METHOD PRIVATE Meth_MororON : BOOL
VAR_INPUT
	Execute: 	BOOL;
END_VAR


	THIS^.Monitoring.StepMessage			:= 'Motor ON';
	THIS^.Monitoring.Error_Text				:= ' Motor ON Fail';
	//THIS^.CMD.Deacivate_Sequence_Time_Out	:= TRUE;	// Disable time out to the all sequence
	THIS^.CMD.DeactivateStepTimeOut			:= TRUE;	// Disable time out to the actual step
	THIS^.Parameter.TimeOut					:= T#5S;


											
	THIS^.Delay.IN:=TRUE;
	THIS^.Delay.PT :=DINT_TO_TIME( Persist.PersistentStruct.TimerMotorOn);// Ctrl_ref.Parameters.TimerPressDown1);
	IF THIS^.Delay.Q  AND FB_RW_Ctrl_ref.Done THEN
		Meth_MororON	:= TRUE;
	END_IF
END_METHOD

METHOD Meth_OutGripperClamp : BOOL
VAR_INPUT
	Execute: 	BOOL;
END_VAR


	THIS^.Monitoring.StepMessage			:= 'Output Gripper Close';
	THIS^.Monitoring.Error_Text				:= ' Fail';
	//THIS^.CMD.Deacivate_Sequence_Time_Out	:= TRUE;	// Disable time out to the all sequence
	THIS^.CMD.DeactivateStepTimeOut			:= TRUE;	// Disable time out to the actual step
	THIS^.Parameter.TimeOut					:= T#5S;

	gMachineCtrl.IO.Out.Output_GripperClose:=TRUE;
											
	THIS^.Delay.IN:=TRUE;
	THIS^.Delay.PT :=DINT_TO_TIME( Persist.PersistentStruct.TimeOutputGripperClose);// Ctrl_ref.Parameters.TimerPressDown1);
	IF THIS^.Delay.Q THEN
		Meth_OutGripperClamp	:= TRUE;
		
		//gMachineCtrl.Parameters.UW_1_Param.EnableTension:=TRUE;
		//gMachineCtrl.Parameters.UW_2_Param.EnableTension:=TRUE;
		
	END_IF
END_METHOD

METHOD Meth_OutGripperEndPos : BOOL
VAR_INPUT
	Execute: 	BOOL;
END_VAR
VAR_INST
	ExecuteTrig: 	Trigger;
END_VAR




IF ExecuteTrig.EDGEPOS(Execute) THEN
	Meth_OutGripperEndPos:=	FALSE;
	THIS^.SubStepNo:= 	1;	
END_IF

IF ExecuteTrig.EDGENEG(Execute) THEN
	Meth_OutGripperEndPos:=	FALSE;
END_IF

CASE THIS^.SubStepNo OF
	(* Power ON*)
	1:
		THIS^.Monitoring.StepMessage	:= 'Move output gripper to end';								
		gWebAxes.Output.Crtl.Basic_axis.Input.Command.MoveAbsolute		:= TRUE;
		gWebAxes.Output.Crtl.Basic_axis.Input.Parameter.Velocity		:= 500;//mm/sec
		gWebAxes.Output.Crtl.Basic_axis.Input.Parameter.Position		:= gMachineCtrl.Parameters.OutgripperEndPosition;//mm
		
		THIS^.SubStepNo:= 2;		
	
	2:	
		THIS^.Monitoring.StepMessage:= 'Wait output gripper end';
		
		IF gWebAxes.Output.Crtl.Basic_axis.Output.monitor.ActPosition > (gMachineCtrl.Parameters.OutgripperEndPosition-200) THEN
			gMachineCtrl.IO.Out.Output_GripperClose:=FALSE;
		END_IF
							
		IF gWebAxes.Output.Crtl.Basic_axis.Output.Status.MC_MoveAbsolut.Done THEN
			THIS^.SubStepNo	:= 3 ;
		END_IF
		
	3:	
		THIS^.Monitoring.StepMessage	:= 'Move output gripper to end';								
		gWebAxes.Output.Crtl.Basic_axis.Input.Command.MoveAbsolute		:= TRUE;
		gWebAxes.Output.Crtl.Basic_axis.Input.Parameter.Velocity		:= 100;//mm/sec
		gWebAxes.Output.Crtl.Basic_axis.Input.Parameter.Position		:= gMachineCtrl.Parameters.OutgripperEndPosition+200;//mm
		
		THIS^.SubStepNo:= 4;	
				
	4:	
		THIS^.Monitoring.StepMessage:= 'Wait output gripper end';
							
		IF gWebAxes.Output.Crtl.Basic_axis.Output.Status.MC_MoveAbsolut.Done THEN
			THIS^.SubStepNo	:= 100 ;
			Meth_OutGripperEndPos:=	TRUE;
		END_IF							
END_CASE
END_METHOD

METHOD Meth_OutGripperStartPos : BOOL
VAR_INPUT
	Execute: 	BOOL;
END_VAR
VAR_INST
	ExecuteTrig: 	Trigger;
END_VAR




IF ExecuteTrig.EDGEPOS(Execute) THEN
	Meth_OutGripperStartPos:=	FALSE;
	THIS^.SubStepNo:= 	1;	
END_IF

IF ExecuteTrig.EDGENEG(Execute) THEN
	Meth_OutGripperStartPos:=	FALSE;
END_IF

CASE THIS^.SubStepNo OF
	(* Power ON*)
	1:
		THIS^.Monitoring.StepMessage	:= 'Move output gripper to home';								
		gWebAxes.Output.Crtl.Basic_axis.Input.Command.MoveAbsolute		:= TRUE;
		gWebAxes.Output.Crtl.Basic_axis.Input.Parameter.Velocity		:= 500;//mm/sec
		gWebAxes.Output.Crtl.Basic_axis.Input.Parameter.Position		:= 0;
		
		THIS^.SubStepNo:= 2;		
	
	2:	
		THIS^.Monitoring.StepMessage:= 'Wait output gripper home';
									
		IF gWebAxes.Output.Crtl.Basic_axis.Output.Status.MC_MoveAbsolut.Done THEN
			THIS^.SubStepNo	:= 3 ;
			Meth_OutGripperStartPos	:= TRUE;
		END_IF
		

							
END_CASE
END_METHOD

METHOD Meth_Rest_IO 
VAR_INPUT
	
END_VAR

Ctrl_ref.IO.Out.HeaterOn := FALSE;
END_METHOD

METHOD PRIVATE Meth_WaitDancerFull : BOOL
VAR_INPUT
	Execute: 	BOOL;
END_VAR


	//THIS^.Monitoring.StepMessage			:= 'Gripper Retract';
	THIS^.Monitoring.Error_Text				:= ' Fail';
	//THIS^.CMD.Deacivate_Sequence_Time_Out	:= TRUE;	// Disable time out to the all sequence
	THIS^.CMD.DeactivateStepTimeOut			:= TRUE;	// Disable time out to the actual step
	THIS^.Parameter.TimeOut					:= T#5S;

	gMachineCtrl.Parameters.UW_1_Param.EnableDancer :=TRUE;
	gMachineCtrl.Parameters.UW_2_Param.EnableDancer:=TRUE;
											
	THIS^.Delay.IN:=TRUE;
	THIS^.Delay.PT :=DINT_TO_TIME( Persist.PersistentStruct.TimeGripperRetract);// Ctrl_ref.Parameters.TimerPressDown1);
	IF  (gMachineCtrl.Status.UW_1_DancerFull 
	AND gMachineCtrl.Status.UW_2_DancerFull)
	OR gMachineCtrl.Simulation THEN
		Meth_WaitDancerFull	:= TRUE;
	END_IF
END_METHOD

END_FUNCTION_BLOCK

// ---- POUs/App/FB_HeaterProtection.TcPOU
FUNCTION_BLOCK FB_HeaterProtection
VAR_INPUT
	Excute:BOOL;
END_VAR
VAR_OUTPUT
	Done:BOOL;
	Busy:BOOL;
END_VAR
VAR
	Timer:TON;
	Step:INT;
END_VAR


IF Excute THEN
	Step:= 10;
	Done:=FALSE;
	Excute:=FALSE;
	Busy:=TRUE;
	
	
END_IF

CASE Step OF

	0://wait
	
	10:
		Timer.PT := DINT_TO_TIME( Persist.PersistentStruct.TimerHotWeldingOn);
		Timer.IN:=TRUE;
		gMachineCtrl.IO.Out.HeaterOn:=TRUE;
		IF Timer.Q THEN
			gMachineCtrl.IO.Out.HeaterOn:=FALSE;
			Step:=20;
		END_IF
	
	20:
		Done:=TRUE;
		Timer.IN:=FALSE;
		Busy:=FALSE;
	
END_CASE

Timer();

END_FUNCTION_BLOCK

// ---- POUs/App/FB_Mechinit.TcPOU
FUNCTION_BLOCK FB_Mechinit EXTENDS CycleHandleFB
VAR_INPUT
	Ctrl_ref:			REFERENCE TO Ctrl_Typ;
END_VAR
VAR_OUTPUT
END_VAR
VAR
	MethInitDone:		BOOL;
END_VAR

VAR CONSTANT
// States are global
		
	MECHINIT_INIT:							INT:=0;
	MECHINIT_SWITCH_ON:						INT:=10;
	MECHINIT_RUN_MASTER:					INT:=20;
	MECHINIT_GEAR_IN:						INT:=30;
	MECHINIT_DONE:							INT:=100;
END_VAR

	IF NOT MethInitDone THEN
		MethInitDone	:= Meth_Init();
	END_IF
	
	IF  THIS^.CMD.Pause = FALSE THEN
		
		//-----------------------------
		//State Machine
		//-----------------------------
		CASE THIS^.StepNo OF
			MECHINIT_INIT:
				IF THIS^.StepOneShotTrig THEN
					THIS^.Monitoring.StepMessage	:= 'Init: Start.';
					THIS^.Delay(IN:=FALSE);
				ELSIF Meth_Enable(TRUE) THEN
					THIS^.StepNo	:= 	MECHINIT_SWITCH_ON;
				END_IF
			
			MECHINIT_SWITCH_ON:
				IF THIS^.StepOneShotTrig THEN
					THIS^.Monitoring.StepMessage	:= 'Switch motor on.';
					THIS^.Delay(IN:=FALSE);
					Meth_SwitchOn(FALSE);
				ELSIF Meth_SwitchOn(TRUE) THEN
					THIS^.StepNo	:= 	MECHINIT_RUN_MASTER;
				END_IF	
				
			MECHINIT_RUN_MASTER:
				IF THIS^.StepOneShotTrig THEN
					THIS^.Monitoring.StepMessage	:= 'Start master';
					THIS^.Delay(IN:=FALSE);
					Meth_StartVmaster(FALSE);
				ELSIF Meth_StartVmaster(TRUE) THEN
					THIS^.StepNo	:= 	MECHINIT_GEAR_IN;
				END_IF				
				

			MECHINIT_GEAR_IN:
				IF THIS^.StepOneShotTrig THEN
					THIS^.Monitoring.StepMessage	:= 'Gear In';
					THIS^.Delay(IN:=FALSE);
					Meth_GearIn(FALSE);
				ELSIF Meth_GearIn(TRUE) THEN
					THIS^.StepNo	:= 	MECHINIT_DONE;
				END_IF	
				
				
			MECHINIT_DONE:
				IF THIS^.StepOneShotTrig THEN
					THIS^.Monitoring.StepMessage	:= 'mechinit cycle Done';
				ELSIF Meth_Done(TRUE) THEN
					THIS^.StepNo	:= 	MECHINIT_INIT;
				END_IF					
				
		END_CASE
	
	ELSE
		THIS^.Monitoring.StepMessage:= 'Pause';
		
		IF THIS^.Status.Fault = TRUE THEN
		//IF Meth_EmStop(TRUE) THEN
				THIS^.CMD.ResetCycle	:= TRUE;		// Reset the all state machine to start point
		//END_IF
			
		END_IF
		
	END_IF
	
	THIS^.Delay();
	THIS^.CH_Logic();
	
	// Reset Meth_EmStop when at Init State
	IF THIS^.Pause = FALSE THEN
		//Meth_EmStop(FALSE);
	END_IF

METHOD PRIVATE Meth_Done : BOOL
VAR_INPUT
	Execute: 	BOOL;
END_VAR


	//THIS^.Monitoring.StepMessage			:= 'Press 1 engage';
	//THIS^.Monitoring.Error_Text				:= 'Press 1 engage Fail';
	//THIS^.CMD.Deacivate_Sequence_Time_Out	:= TRUE;	// Disable time out to the all sequence
	//THIS^.CMD.DeactivateStepTimeOut			:= TRUE;	// Disable time out to the actual step
	//THIS^.Parameter.TimeOut					:= T#5S;

	THIS^.Status.Done		:= TRUE;
	THIS^.Status.Running	:= FALSE;									
	Meth_Done	:= TRUE;
END_METHOD

METHOD PRIVATE Meth_Enable : BOOL
VAR_INPUT
	Execute: 	BOOL;
END_VAR


IF THIS^.CMD.Start THEN
	
	THIS^.Monitoring.StepMessage			:= 'Start';
	THIS^.Monitoring.Error_Text				:= 'Start Fail';
	THIS^.CMD.Deacivate_Sequence_Time_Out	:= TRUE;	// Disable time out to the all sequence
	THIS^.CMD.DeactivateStepTimeOut			:= TRUE;	// Disable time out to the actual step
	THIS^.Parameter.TimeOut					:= T#0.5S;

	THIS^.CMD.Start			:= FALSE;
	THIS^.Status.Done		:= FALSE;
	THIS^.Status.Running	:= TRUE;
	
	// Reset Commands and Statuses												
	
	Meth_Enable	:= TRUE;
END_IF
END_METHOD

METHOD Meth_GearIn : BOOL
VAR_INPUT
	Execute: 	BOOL;
END_VAR
VAR_INST	
	ExecuteTrig: 	Trigger;	
END_VAR
IF ExecuteTrig.EDGEPOS(Execute) THEN
	Meth_GearIn	:= FALSE;
	THIS^.SubStepNo:= 	1;	
END_IF

IF ExecuteTrig.EDGENEG(Execute) THEN
	Meth_GearIn	:=	FALSE;
END_IF

CASE THIS^.SubStepNo OF
	   
	1:
		THIS^.Monitoring.StepMessage:= 'Set GearInMultiMaster command';
		
		gWebAxes.UW_1.Crtl.MultiAxis.Input.Parameter.GearInMultiMaster.GearRatio1:=	0;

		
		gWebAxes.UW_1.Crtl.MultiAxis.Input.Parameter.GearInMultiMaster.Acceleration:= 	600000;
		gWebAxes.UW_1.Crtl.MultiAxis.Input.Parameter.GearInMultiMaster.Deceleration:= 	600000;
		gWebAxes.UW_1.Crtl.MultiAxis.Input.Parameter.GearInMultiMaster.Jerk:=			0;
		gWebAxes.UW_1.Crtl.MultiAxis.Input.Parameter.GearInMultiMaster.Options.AdvancedSlaveDynamics:= 	FALSE;
		
		gWebAxes.UW_1.Crtl.MultiAxis.Input.Command.GearInMultiMaster.StartSlave:=		TRUE;
				
								
		THIS^.SubStepNo	:= 2;		
			
	2:	
		THIS^.Monitoring.StepMessage:= 	'Wait for GearInMultiMaster done UW1' ;
							
		IF (gWebAxes.UW_1.Crtl.MultiAxis.Input.Command.GearInMultiMaster.StartSlave = FALSE) 
			AND (gWebAxes.UW_1.Crtl.MultiAxis.Output.Status.GearInMultiMaster.InGear = TRUE) THEN
			THIS^.SubStepNo:=	3;
		ELSIF 	gWebAxes.UW_1.Crtl.MultiAxis.Output.Status.GearInMultiMaster.InGear = TRUE THEN
			THIS^.SubStepNo:=	3;
		END_IF		


	3:
		THIS^.Monitoring.StepMessage:= 'Set GearInMultiMaster UW2 command';
		
		gWebAxes.UW_2.Crtl.MultiAxis.Input.Parameter.GearInMultiMaster.GearRatio1:=	0;

		
		gWebAxes.UW_2.Crtl.MultiAxis.Input.Parameter.GearInMultiMaster.Acceleration:= 	600000;
		gWebAxes.UW_2.Crtl.MultiAxis.Input.Parameter.GearInMultiMaster.Deceleration:= 	600000;
		gWebAxes.UW_2.Crtl.MultiAxis.Input.Parameter.GearInMultiMaster.Jerk:=			0;
		gWebAxes.UW_2.Crtl.MultiAxis.Input.Parameter.GearInMultiMaster.Options.AdvancedSlaveDynamics:= 	FALSE;
		
		gWebAxes.UW_2.Crtl.MultiAxis.Input.Command.GearInMultiMaster.StartSlave:=		TRUE;
				
								
		THIS^.SubStepNo	:= 4;		
			
	4:	
		THIS^.Monitoring.StepMessage:= 	'Wait for GearInMultiMaster done' ;
							
		IF (gWebAxes.UW_2.Crtl.MultiAxis.Input.Command.GearInMultiMaster.StartSlave = FALSE) 
			AND (gWebAxes.UW_2.Crtl.MultiAxis.Output.Status.GearInMultiMaster.InGear = TRUE) THEN
			THIS^.SubStepNo:=	0;
			Meth_GearIn:= 	TRUE;
		ELSIF gWebAxes.UW_2.Crtl.MultiAxis.Output.Status.GearInMultiMaster.InGear = TRUE THEN	
			THIS^.SubStepNo:=	0;
			Meth_GearIn:= 	TRUE;
		END_IF	

							
END_CASE
END_METHOD

METHOD Meth_Init :BOOL
VAR_INPUT
END_VAR
//resets


Meth_Init:=TRUE;
END_METHOD

METHOD Meth_StartVmaster : BOOL
VAR_INPUT
	Execute: 	BOOL;
END_VAR
VAR_INST	
	ExecuteTrig: 	Trigger;	
END_VAR

IF ExecuteTrig.EDGEPOS(Execute) THEN
	Meth_StartVmaster	:= FALSE;
	THIS^.SubStepNo:= 	1;	
END_IF

IF ExecuteTrig.EDGENEG(Execute) THEN
	Meth_StartVmaster	:=	FALSE;
END_IF


CASE THIS^.SubStepNo OF
	   
	1:
		THIS^.Monitoring.StepMessage	:= 'Set RunVel command to Master Tension';
		
			gWebAxes.UwVmaster.Crtl.Basic_axis.Input.Parameter.Acceleration	:= 100000; 
			gWebAxes.UwVmaster.Crtl.Basic_axis.Input.Parameter.Deceleration	:= 100000; 
			gWebAxes.UwVmaster.Crtl.Basic_axis.Input.Parameter.Velocity		:= 360000;//100000 
			gWebAxes.UwVmaster.Crtl.Basic_axis.Input.Parameter.Direction		:= MC_Positive_Direction; 		
				
			gWebAxes.UwVmaster.Crtl.Basic_axis.Input.Command.MoveVelocity		:= TRUE;
			THIS^.SubStepNo:= 	2;	

	2:	
		THIS^.Monitoring.StepMessage	:= 'Wait @ velocity from Master';
		IF (gWebAxes.UwVmaster.Crtl.Basic_axis.Output.Status.AxisStatus.ContinuousMotion = TRUE) THEN	
			Meth_StartVmaster:=TRUE;
			THIS^.SubStepNo:= 	0;				
		END_IF
								
END_CASE
END_METHOD

METHOD Meth_SwitchOn : BOOL
VAR_INPUT
	Execute: 	BOOL;
END_VAR
VAR_INST
	ExecuteTrig: 	Trigger;
END_VAR


IF ExecuteTrig.EDGEPOS(Execute) THEN
	Meth_SwitchOn:=	FALSE;
	THIS^.SubStepNo:= 	1;	
END_IF

IF ExecuteTrig.EDGENEG(Execute) THEN
	Meth_SwitchOn:=	FALSE;
END_IF

CASE THIS^.SubStepNo OF
	(* Power ON*)
	1:
		THIS^.Monitoring.StepMessage	:= 'Power On';								
		gWebAxes.UW_1.Crtl.Basic_axis.Input.Command.Power		:= TRUE;
		gWebAxes.UW_2.Crtl.Basic_axis.Input.Command.Power		:= TRUE;	
		gWebAxes.UwVmaster.Crtl.Basic_axis.Input.Command.Power	:= TRUE;
		
		THIS^.SubStepNo:= 2;		
	
	2:	
		THIS^.Monitoring.StepMessage:= 'Wait for standstill UW 1';
									
		IF gWebAxes.UW_1.Crtl.Basic_axis.Output.Status.AxisStatus.StandStill
		OR gWebAxes.UW_1.Crtl.Basic_axis.Output.Status.AxisStatus.SynchronizedMotion THEN
			THIS^.SubStepNo	:= 3 ;
		END_IF
		
	3:	
		THIS^.Monitoring.StepMessage:= 'Wait for standstill UW 2';
									
		IF gWebAxes.UW_2.Crtl.Basic_axis.Output.Status.AxisStatus.StandStill
		OR  gWebAxes.UW_2.Crtl.Basic_axis.Output.Status.AxisStatus.SynchronizedMotion THEN
			THIS^.SubStepNo	:= 4 ;
		END_IF		
		
	4:	
		THIS^.Monitoring.StepMessage:= 'Wait for standstill from master';
									
		IF gWebAxes.UwVmaster.Crtl.Basic_axis.Output.Status.AxisStatus.StandStill
		OR  gWebAxes.UwVmaster.Crtl.Basic_axis.Output.Status.AxisStatus.ContinuousMotion THEN
			THIS^.SubStepNo	:= 10 ;
			Meth_SwitchOn	:= TRUE;
		END_IF
							
END_CASE
END_METHOD

END_FUNCTION_BLOCK

// ---- POUs/App/FB_Machine_Ctrl.TcPOU
FUNCTION_BLOCK FB_Machine_Ctrl EXTENDS CycleHandleFB
VAR_INPUT
	Ctrl_ref:					REFERENCE TO Ctrl_Typ;
	FB_Machine_Run_ref:			REFERENCE TO FB_Machine_Run;
	FB_Mechinit_ref:			REFERENCE TO FB_Mechinit;
	FB_MechinitOutput_ref:		REFERENCE TO FB_MechinitOutput;
	FB_OFF_ref:					REFERENCE TO FB_OFF;
END_VAR
VAR_OUTPUT
END_VAR
VAR
	MethInitDone:		BOOL;
	StopFlag:BOOL;
	
	TriggerOff:Trigger;
	
END_VAR
VAR CONSTANT

// States		
	MAIN_INIT:						INT:=0;
	MAIN_OFF:						INT:=10;
	MAIN_STANDBY:					INT:=11;
	MAIN_MECHINIT:					INT:=15;
	MAIN_RUN:						INT:=20;
	MAIN_EM_STOP:					INT:=100;


END_VAR

	IF NOT MethInitDone THEN
		MethInitDone	:= Meth_Init();
	END_IF
	
	
	IF (gMachineCtrl.Cmd.EmStop)
	AND FB_OFF_ref.Running = FALSE THEN	
		THIS^.StepNo	:= 	MAIN_EM_STOP;
	END_IF
	
	IF  THIS^.CMD.Pause = FALSE THEN
		
		//-----------------------------
		//State Machine
		//-----------------------------
		CASE THIS^.StepNo OF
			MAIN_INIT:
				IF THIS^.StepOneShotTrig THEN
					THIS^.Monitoring.StepMessage	:= 'Init: Start.';
				ELSIF Meth_Enable(TRUE) THEN
					THIS^.StepNo	:= 	MAIN_OFF;
				END_IF
			
			MAIN_OFF:
				IF THIS^.StepOneShotTrig THEN
					THIS^.Monitoring.StepMessage	:= 'OFF';
				ELSIF Meth_Standby(TRUE) THEN
					THIS^.StepNo	:= 	MAIN_MECHINIT;
				END_IF
				
			MAIN_MECHINIT:
				IF THIS^.StepOneShotTrig THEN
					THIS^.Monitoring.StepMessage	:= 'Mechinit';
					Meth_Mechint(FALSE);
				ELSIF Meth_Mechint(TRUE) THEN
					THIS^.StepNo	:= 	MAIN_STANDBY;
				END_IF				

	
			MAIN_STANDBY:
				IF THIS^.StepOneShotTrig THEN
					THIS^.Monitoring.StepMessage	:= 'OFF';
				ELSIF Meth_Start(TRUE) THEN
					THIS^.StepNo	:= 	MAIN_RUN;
				END_IF				
			
			
				
			MAIN_RUN:
				IF THIS^.StepOneShotTrig THEN
					THIS^.Monitoring.StepMessage	:= 'RUN';
					Meth_Run(FALSE);
				ELSIF Meth_Run(TRUE) THEN
					THIS^.StepNo	:= 	MAIN_INIT;
				END_IF
	
				
			//OFF
			MAIN_EM_STOP:
				IF THIS^.StepOneShotTrig THEN
					THIS^.Monitoring.StepMessage	:= 'Powering OFF';
					Meth_EmStop(FALSE);
				ELSIF Meth_EmStop(TRUE) THEN
					THIS^.StepNo	:= 	MAIN_INIT;
				END_IF				
				
		END_CASE
	
	ELSE
		THIS^.Monitoring.StepMessage:= 'Pause';
		
		IF THIS^.Status.Fault = TRUE THEN
			IF Meth_EmStop(TRUE) THEN
				THIS^.CMD.ResetCycle	:= TRUE;		// Reset the all state machine to start point
			END_IF
			
		END_IF
		
	END_IF
	

	
	// Reset Meth_EmStop when at Init State
	//IF THIS^.Pause = FALSE THEN
	//	Meth_EmStop(FALSE);
	//END_IF
	
	
	(*
	
	
	//============================================================================================
	// Any Fb Fault
	AnyFbFaultFlag	:= fbMechInit_ref.Fault OR fbRun_ref.Fault OR fbStop_ref.Fault;
	
	//============================================================================================
	// Set Fault flag on bEmStopActive_ref or bExternalFault
	IF (THIS^.Status.Running = TRUE)
		AND (ExternalFaultTrig.EDGEPOS(bExternalFault)
			OR EmStopTrig.EDGEPOS(bEmStopActive_ref
				AND Ctrl_ref.Out.Status.InitDone
				AND Ctrl_ref.Out.Status.AtPowerDisable = FALSE
				AND Ctrl_ref.Out.Status.AtOff = FALSE)
			OR AnyFbFaultFlag)  THEN
		THIS^.Fault	:= TRUE;	// When fault, Pause rise automatic on the fb
	END_IF
	
	
	
	*)
	//============================================================================================
	// Reset Internal Function Blocks
	IF THIS^.CMD.ResetCycle = TRUE THEN
		IF FB_Machine_Run_ref.Running OR FB_Machine_Run_ref.Pause OR FB_Machine_Run_ref.Fault THEN
			FB_Machine_Run_ref.ResetCycle	:= TRUE;
		END_IF
	END_IF
	
	//============================================================================================			
	
	
THIS^.Delay();
THIS^.CH_Logic();

METHOD Meth_EmStop : BOOL
VAR_INPUT
	Execute: 	BOOL;
END_VAR

VAR_INST	
	ExecuteTrig: 	Trigger;	
END_VAR


IF ExecuteTrig.EDGEPOS(Execute) THEN
	Meth_EmStop	:= FALSE;
	THIS^.SubStepNo:= 	1;	
END_IF

IF ExecuteTrig.EDGENEG(Execute) THEN
	Meth_EmStop	:=	FALSE;
END_IF

gMachineCtrl.Cmd.EmStop:=FALSE;

CASE THIS^.SubStepNo OF
	   
	1:
		//THIS^.Monitoring.StepMessage	:= 'Start mechint';
		THIS^.FB_OFF_ref.Start	:=TRUE;
		THIS^.SubStepNo:=2;
		
	2:
		//THIS^.Monitoring.StepMessage	:= 'Wait  Mechint';
		IF THIS^.FB_OFF_ref.Done	THEN
			THIS^.SubStepNo:=0;
			Meth_EmStop	:=	TRUE;
		END_IF
	
END_CASE
END_METHOD

METHOD PRIVATE Meth_Enable : BOOL
VAR_INPUT
	Execute: 	BOOL;
END_VAR

IF MethInitDone then
	THIS^.CMD.Start	:= TRUE;
END_IF

IF THIS^.CMD.Start THEN
	
	THIS^.Monitoring.StepMessage			:= 'Start';
	THIS^.Monitoring.Error_Text				:= 'Start Fail';
	THIS^.CMD.Deacivate_Sequence_Time_Out	:= TRUE;	// Disable time out to the all sequence
	THIS^.CMD.DeactivateStepTimeOut			:= TRUE;	// Disable time out to the actual step
	THIS^.Parameter.TimeOut					:= T#0.5S;

	THIS^.CMD.Start			:= FALSE;
	THIS^.Status.Done		:= FALSE;
	THIS^.Status.Running	:= TRUE;
	
	// Reset Commands and Statuses												
	
	Meth_Enable	:= TRUE;
END_IF
END_METHOD

METHOD Meth_Init :BOOL
VAR_INPUT
END_VAR
Meth_Init:=TRUE;
END_METHOD

METHOD Meth_Mechint : BOOL
VAR_INPUT
	Execute:BOOL;
END_VAR
VAR_INST	
	ExecuteTrig: 	Trigger;	
END_VAR

IF ExecuteTrig.EDGEPOS(Execute) THEN
	Meth_Mechint	:= FALSE;
	THIS^.SubStepNo:= 	1;	
END_IF

IF ExecuteTrig.EDGENEG(Execute) THEN
	Meth_Mechint	:=	FALSE;
END_IF

CASE THIS^.SubStepNo OF
	   
	1:
		THIS^.Monitoring.StepMessage		:= 'Start mechint';
		THIS^.FB_Mechinit_ref.Start			:=TRUE;
		THIS^.FB_MechinitOutput_ref.Start	:=TRUE;		
		THIS^.SubStepNo:=2;
		
	2:
		THIS^.Monitoring.StepMessage	:= 'Wait  Mechint Output';
		IF THIS^.FB_MechinitOutput_ref.Done	THEN
			THIS^.SubStepNo:=3;
		END_IF
	3:
		THIS^.Monitoring.StepMessage	:= 'Wait  Mechint Input';
		IF THIS^.FB_Mechinit_ref.Done	THEN
			THIS^.SubStepNo:=0;
			Meth_Mechint	:=	TRUE;
		END_IF	
END_CASE
END_METHOD

METHOD Meth_Run : BOOL;
VAR_INPUT
	Excute:BOOL;
END_VAR

IF Excute = FALSE THEN
	THIS^.SubStepNo :=0;
ELSIF Excute AND_THEN THIS^.SubStepNo = 0 THEN
	THIS^.SubStepNo :=10;
END_IF	

IF Ctrl_ref.Cmd.Stop THEN
	StopFlag:=TRUE;
	THIS^.Monitoring.StepMessage	:= 'STOPPING';
END_IF


CASE THIS^.SubStepNo OF
	
	0://Wait
		THIS^.Monitoring.SubStepMessage	:= 'Wait';
		
	10://Start
		THIS^.Monitoring.SubStepMessage	:= 'Statr';	
		FB_Machine_Run_ref.Start	 :=TRUE;
		THIS^.SubStepNo				:=20;
		
	20://Wait cycle end	
		THIS^.Monitoring.SubStepMessage	:= 'Wait cycle to end';	
		IF FB_Machine_Run_ref.Done THEN
			THIS^.SubStepNo				:=30;
			Ctrl_ref.Status.SessionCounter:=Ctrl_ref.Status.SessionCounter+1;
			PersistentStruct.LifeTimerCounter:=PersistentStruct.LifeTimerCounter+1;
		END_IF
	
	30: //Check if continue	or Stop
		IF StopFlag THEN
			Meth_Run :=TRUE;
		ELSIF Ctrl_ref.Parameters.Continues 
		OR Ctrl_ref.Status.SessionCounter < Ctrl_ref.Parameters.NumberOfCycles   THEN
			THIS^.SubStepNo		:=10;
		ELSE
			 Meth_Run :=TRUE;		
		END_IF

END_CASE
END_METHOD

METHOD Meth_Standby : BOOL
VAR_INPUT
	Execute: 	BOOL;
END_VAR

IF Ctrl_ref.Cmd.SwitchOn THEN
	Meth_Standby:=TRUE;
	//Ctrl_ref.Cmd.Start:=FALSE;
	
	//reset session
	//StopFlag:=FALSE;
	//Ctrl_ref.Status.SessionCounter:=0;	
	
ELSIF	Ctrl_ref.Cmd.Manual THEN
	THIS^.Monitoring.StepMessage	:= 'Manual';
ELSE
	THIS^.Monitoring.StepMessage	:= 'OFF';	
END_IF
END_METHOD

METHOD Meth_Start : BOOL
VAR_INPUT
	Execute: 	BOOL;
END_VAR

IF Ctrl_ref.Cmd.Start THEN
	Meth_Start:=TRUE;
	Ctrl_ref.Cmd.Start:=FALSE;
	
	//reset session
	StopFlag:=FALSE;
	Ctrl_ref.Status.SessionCounter:=0;	
	
ELSIF	Ctrl_ref.Cmd.Manual THEN
	THIS^.Monitoring.StepMessage	:= 'Manual';
ELSE
	THIS^.Monitoring.StepMessage	:= 'StandBy';	
END_IF
END_METHOD

END_FUNCTION_BLOCK

// ---- POUs/App/FB_MechinitOutput.TcPOU
FUNCTION_BLOCK FB_MechinitOutput EXTENDS CycleHandleFB
VAR_INPUT
	Ctrl_ref:			REFERENCE TO Ctrl_Typ;
END_VAR
VAR_OUTPUT
END_VAR
VAR
	MethInitDone:		BOOL;
END_VAR

VAR CONSTANT
// States are global
		
	MECHINIT_OUT_INIT:					INT:=0;
	MECHINIT_OUT_SWITCH_ON:				INT:=10;
	MECHINIT_OUT_HOME:					INT:=20;

	MECHINIT_OUT_DONE:					INT:=100;
END_VAR

	IF NOT MethInitDone THEN
		MethInitDone	:= Meth_Init();
	END_IF
	
	IF  THIS^.CMD.Pause = FALSE THEN
		
		//-----------------------------
		//State Machine
		//-----------------------------
		CASE THIS^.StepNo OF
			MECHINIT_OUT_INIT:
				IF THIS^.StepOneShotTrig THEN
					THIS^.Monitoring.StepMessage	:= 'Init: out Start.';
					THIS^.Delay(IN:=FALSE);
				ELSIF Meth_Enable(TRUE) THEN
					THIS^.StepNo	:= 	MECHINIT_OUT_SWITCH_ON;
				END_IF
			
			MECHINIT_OUT_SWITCH_ON:
				IF THIS^.StepOneShotTrig THEN
					THIS^.Monitoring.StepMessage	:= 'Switch motor on.';
					THIS^.Delay(IN:=FALSE);
					Meth_SwitchOn(FALSE);
				ELSIF Meth_SwitchOn(TRUE) THEN
					THIS^.StepNo	:= 	MECHINIT_OUT_HOME;
				END_IF	
				
			MECHINIT_OUT_HOME:
				IF THIS^.StepOneShotTrig THEN
					THIS^.Monitoring.StepMessage	:= 'Home';
					THIS^.Delay(IN:=FALSE);
					Meth_Home(FALSE);
				ELSIF Meth_Home(TRUE) THEN
					THIS^.StepNo	:= 	MECHINIT_OUT_DONE;
				END_IF				
			
				
				
			MECHINIT_OUT_DONE:
				IF THIS^.StepOneShotTrig THEN
					THIS^.Monitoring.StepMessage	:= 'mechinit cycle Done';
				ELSIF Meth_Done(TRUE) THEN
					THIS^.StepNo	:= 	MECHINIT_OUT_INIT;
				END_IF					
				
		END_CASE
	
	ELSE
		THIS^.Monitoring.StepMessage:= 'Pause';
		
		IF THIS^.Status.Fault = TRUE THEN
		//IF Meth_EmStop(TRUE) THEN
				THIS^.CMD.ResetCycle	:= TRUE;		// Reset the all state machine to start point
		//END_IF
			
		END_IF
		
	END_IF
	
	THIS^.Delay();
	THIS^.CH_Logic();
	
	// Reset Meth_EmStop when at Init State
	IF THIS^.Pause = FALSE THEN
		//Meth_EmStop(FALSE);
	END_IF

METHOD PRIVATE Meth_Done : BOOL
VAR_INPUT
	Execute: 	BOOL;
END_VAR


	//THIS^.Monitoring.StepMessage			:= 'Press 1 engage';
	//THIS^.Monitoring.Error_Text				:= 'Press 1 engage Fail';
	//THIS^.CMD.Deacivate_Sequence_Time_Out	:= TRUE;	// Disable time out to the all sequence
	//THIS^.CMD.DeactivateStepTimeOut			:= TRUE;	// Disable time out to the actual step
	//THIS^.Parameter.TimeOut					:= T#5S;

	THIS^.Status.Done		:= TRUE;
	THIS^.Status.Running	:= FALSE;									
	Meth_Done	:= TRUE;
END_METHOD

METHOD PRIVATE Meth_Enable : BOOL
VAR_INPUT
	Execute: 	BOOL;
END_VAR


IF THIS^.CMD.Start THEN
	
	THIS^.Monitoring.StepMessage			:= 'Start output';
	THIS^.Monitoring.Error_Text				:= 'Start Fail';
	THIS^.CMD.Deacivate_Sequence_Time_Out	:= TRUE;	// Disable time out to the all sequence
	THIS^.CMD.DeactivateStepTimeOut			:= TRUE;	// Disable time out to the actual step
	THIS^.Parameter.TimeOut					:= T#0.5S;

	THIS^.CMD.Start			:= FALSE;
	THIS^.Status.Done		:= FALSE;
	THIS^.Status.Running	:= TRUE;
	
	// Reset Commands and Statuses												
	
	Meth_Enable	:= TRUE;
END_IF
END_METHOD

METHOD Meth_Home : BOOL
VAR_INPUT
	Execute: 	BOOL;
END_VAR
VAR_INST
	ExecuteTrig: 	Trigger;
END_VAR


IF ExecuteTrig.EDGEPOS(Execute) THEN
	Meth_Home:=	FALSE;
	THIS^.SubStepNo:= 	1;	
END_IF

IF ExecuteTrig.EDGENEG(Execute) THEN
	Meth_Home:=	FALSE;
END_IF

CASE THIS^.SubStepNo OF
	(* Power ON*)
	1:
		THIS^.Monitoring.StepMessage	:= 'Move Addative';								
		gWebAxes.Output.Crtl.Basic_axis.Input.Command.MoveAdditive		:= TRUE;
		gWebAxes.Output.Crtl.Basic_axis.Input.Parameter.Acceleration	:= 10000;//[mm/sec^2]
		gWebAxes.Output.Crtl.Basic_axis.Input.Parameter.Deceleration	:= 10000;//[mm/sec^2]	
		gWebAxes.Output.Crtl.Basic_axis.Input.Parameter.Distance		:= -2500;//[mm/sec^2]	
		gWebAxes.Output.Crtl.Basic_axis.Input.Parameter.Velocity		:= gMachineCtrl.Parameters.OutGripperHomeVelocity;//[mm/sec]	
		gWebAxes.Output.Crtl.Basic_axis.Input.Parameter.Direction		:= MC_Direction.MC_Positive_Direction;		
		
		THIS^.SubStepNo:= 2;		
	
	2:	
		THIS^.Monitoring.StepMessage:= 'Wait home sensor';
									
		IF gMachineCtrl.IO.In.HomeOutAxis OR gMachineCtrl.Simulation THEN
			gWebAxes.Output.Crtl.Basic_axis.Input.Command.Stop	:= TRUE;
			gWebAxes.Output.Crtl.Basic_axis.Input.Parameter.HomeOptions.stBasic.HomeMode := MC_HomingMode.MC_Direct;
			THIS^.SubStepNo	:= 3 ;
		END_IF
		
	3:	
		THIS^.Monitoring.StepMessage:= 'Wait stop';
		IF gWebAxes.Output.Crtl.Basic_axis.Output.Status.AxisStatus.StandStill THEN
			gWebAxes.Output.Crtl.Basic_axis.Input.Command.Home		:= TRUE;
			THIS^.SubStepNo	:= 4 ;
		END_IF									
	
		
	4:	
		THIS^.Monitoring.StepMessage:= 'wait home done';			
		IF gWebAxes.Output.Crtl.Basic_axis.Output.Status.MC_Home.Done THEN
			THIS^.SubStepNo	:= 10 ;
			Meth_Home	:= TRUE;
		END_IF			
							
END_CASE
END_METHOD

METHOD Meth_Init :BOOL
VAR_INPUT
END_VAR
//resets


Meth_Init:=TRUE;
END_METHOD

METHOD Meth_SwitchOn : BOOL
VAR_INPUT
	Execute: 	BOOL;
END_VAR
VAR_INST
	ExecuteTrig: 	Trigger;
END_VAR


IF ExecuteTrig.EDGEPOS(Execute) THEN
	Meth_SwitchOn:=	FALSE;
	THIS^.SubStepNo:= 	1;	
END_IF

IF ExecuteTrig.EDGENEG(Execute) THEN
	Meth_SwitchOn:=	FALSE;
END_IF

CASE THIS^.SubStepNo OF
	(* Power ON*)
	1:
		THIS^.Monitoring.StepMessage	:= 'Power On';								
		gWebAxes.Output.Crtl.Basic_axis.Input.Command.Power		:= TRUE;
		
		THIS^.SubStepNo:= 2;		
	
	2:	
		THIS^.Monitoring.StepMessage:= 'Wait for standstill output';
									
		IF gWebAxes.Output.Crtl.Basic_axis.Output.Status.AxisStatus.StandStill THEN
			THIS^.SubStepNo	:= 10 ;
			Meth_SwitchOn	:= TRUE;
		END_IF
		
							
END_CASE
END_METHOD

END_FUNCTION_BLOCK

// ---- POUs/prg_Motion.TcPOU
PROGRAM prg_Motion
VAR
	UW_1_Diameter:	Dimeter_Typ;
	UW_2_Diameter:	Dimeter_Typ;
	UW_1_Data	:WinderParam_Typ;
	UW_2_Data	:WinderParam_Typ;
	
	Init:BOOL :=TRUE;
END_VAR

IF Init THEN
	Init:=FALSE;
	ACT_init();
END_IF

ACT_DancerCtrl_1();
ACT_DancerCtrl_2();
ACT_Diameter();
ACT_Tension_1();
ACT_Tension_2();
ACT_GearRatio();
ACT_MotionFBcall();

ACTION ACT_DancerCtrl_1:
////////////UW1
UW_1_Data.Dancer.stLutDataParam.eLutMode	:= E_LutMode.eAnalogToPhisical;

UW_1_Data.Dancer.stLutDataParam.arrAnalog[0]		:= -3700;//-30000;
UW_1_Data.Dancer.stLutDataParam.arrPhisical[0]		:= 0;//11000;	//[Dummy]
UW_1_Data.Dancer.stLutDataParam.arrAnalog[1]		:= 12700;//-11500;
UW_1_Data.Dancer.stLutDataParam.arrPhisical[1]		:= 300;//10000;	//[gram]	
UW_1_Data.Dancer.stLutDataParam.arrAnalog[2]		:= 35500;//-600;
UW_1_Data.Dancer.stLutDataParam.arrPhisical[2]		:= 700;//0;	//[gram]	
UW_1_Data.Dancer.stLutDataParam.arrAnalog[3]		:= 65535;//20000;
UW_1_Data.Dancer.stLutDataParam.arrPhisical[3]		:= 1500;//2000;	//[Dummy]

UW_1_Data.Dancer.DancerPosition_Unfiltred
			:= LookUP_Table(RawValue:=gMachineCtrl.IO.In.UW_1_DancerPosition,pDataParam:= ADR(UW_1_Data.Dancer.stLutDataParam));	

UW_1_Data.Dancer.DancerLPF(IN:=UW_1_Data.Dancer.DancerPosition_Unfiltred,out=> UW_1_Data.Dancer.DancerPosition_filtred);

UW_1_Data.Dancer.fb_DancerCtrl.Enable 			:= gMachineCtrl.Parameters.UW_1_Param.EnableDancer;
UW_1_Data.Dancer.fb_DancerCtrl.DancerFull		:= gMachineCtrl.IO.In.UW_1_DancerFull;
UW_1_Data.Dancer.fb_DancerCtrl.DancerPosition	:= UW_1_Data.Dancer.DancerPosition_filtred;
UW_1_Data.Dancer.fb_DancerCtrl.Ctrl_Type		:= E_DancerCtrlTyp.DIGITAL;
UW_1_Data.Dancer.fb_DancerCtrl();
//Connect to jog cmd
gMachineCtrl.Cmd.UW_1_Cmd.JogDancerFill	:= UW_1_Data.Dancer.fb_DancerCtrl.Jog;
gMachineCtrl.Status.UW_1_DancerFull		:= UW_1_Data.Dancer.fb_DancerCtrl.dancerFullStatus;

IF gMachineCtrl.Cmd.UW_1_Cmd.JogDancerFill  THEN
	UW_1_Data.Dancer.DancerGear := gMachineCtrl.Parameters.DancerFillSpeed/360000;
ELSE
	UW_1_Data.Dancer.DancerGear := 0;
END_IF
END_ACTION

ACTION ACT_DancerCtrl_2:
////////////UW1
UW_2_Data.Dancer.stLutDataParam.eLutMode	:= E_LutMode.eAnalogToPhisical;

UW_2_Data.Dancer.stLutDataParam.arrAnalog[0]		:= -3700;//-30000;
UW_2_Data.Dancer.stLutDataParam.arrPhisical[0]		:= 0;//11000;	//[Dummy]
UW_2_Data.Dancer.stLutDataParam.arrAnalog[1]		:= 12700;//-11500;
UW_2_Data.Dancer.stLutDataParam.arrPhisical[1]		:= 300;//10000;	//[gram]	
UW_2_Data.Dancer.stLutDataParam.arrAnalog[2]		:= 35500;//-600;
UW_2_Data.Dancer.stLutDataParam.arrPhisical[2]		:= 700;//0;	//[gram]	
UW_2_Data.Dancer.stLutDataParam.arrAnalog[3]		:= 65535;//20000;
UW_2_Data.Dancer.stLutDataParam.arrPhisical[3]		:= 1500;//2000;	//[Dummy]

UW_2_Data.Dancer.DancerPosition_Unfiltred
			:= LookUP_Table(RawValue:=gMachineCtrl.IO.In.UW_2_DancerPosition,pDataParam:= ADR(UW_2_Data.Dancer.stLutDataParam));	

UW_2_Data.Dancer.DancerLPF(IN:=UW_2_Data.Dancer.DancerPosition_Unfiltred,out=> UW_2_Data.Dancer.DancerPosition_filtred);

UW_2_Data.Dancer.fb_DancerCtrl.Enable 			:= gMachineCtrl.Parameters.UW_2_Param.EnableDancer;
UW_2_Data.Dancer.fb_DancerCtrl.DancerFull		:= gMachineCtrl.IO.In.UW_2_DancerFull;
UW_2_Data.Dancer.fb_DancerCtrl.DancerPosition	:= UW_2_Data.Dancer.DancerPosition_filtred;
UW_2_Data.Dancer.fb_DancerCtrl.Ctrl_Type		:= E_DancerCtrlTyp.DIGITAL;
UW_2_Data.Dancer.fb_DancerCtrl();
//Connect to jog cmd
gMachineCtrl.Cmd.UW_2_Cmd.JogDancerFill	:= UW_2_Data.Dancer.fb_DancerCtrl.Jog;
gMachineCtrl.Status.UW_2_DancerFull		:= UW_2_Data.Dancer.fb_DancerCtrl.dancerFullStatus;

IF gMachineCtrl.Cmd.UW_2_Cmd.JogDancerFill  THEN
	UW_2_Data.Dancer.DancerGear := gMachineCtrl.Parameters.DancerFillSpeed/360000;
ELSE
	UW_2_Data.Dancer.DancerGear := 0;
END_IF
END_ACTION

ACTION ACT_Diameter:

////////////UW1
UW_1_Diameter.stLutDataParam.eLutMode	:= E_LutMode.eAnalogToPhisical;

UW_1_Diameter.stLutDataParam.arrAnalog[0]		:= 0;
UW_1_Diameter.stLutDataParam.arrPhisical[0]		:= 200;	//[mm]
UW_1_Diameter.stLutDataParam.arrAnalog[1]		:= 2600;
UW_1_Diameter.stLutDataParam.arrPhisical[1]		:= 355;	//[mm]	
UW_1_Diameter.stLutDataParam.arrAnalog[2]		:= 7500;
UW_1_Diameter.stLutDataParam.arrPhisical[2]		:= 97;	//[mm]	
UW_1_Diameter.stLutDataParam.arrAnalog[3]		:= 32000;
UW_1_Diameter.stLutDataParam.arrPhisical[3]		:= 0;	

UW_1_Diameter.Diameter_Unfiltred 
			:= LookUP_Table(RawValue:=gMachineCtrl.IO.In.UW_1_Diameter,pDataParam:= ADR(UW_1_Diameter.stLutDataParam));	
			
//UW_1_Diameter.DiameterLPF.IN := UW_1_Diameter.Diameter_Unfiltred;

IF gMachineCtrl.Parameters.UW_1_Param.ForceDiameter THEN
	UW_1_Diameter.Diameter_filtred := gMachineCtrl.Parameters.UW_1_Param.ForcedDiameter;
ELSE
	UW_1_Diameter.DiameterLPF(IN:=UW_1_Diameter.Diameter_Unfiltred,out=> UW_1_Diameter.Diameter_filtred);	
END_IF	

///////////UW2
UW_2_Diameter.stLutDataParam.eLutMode	:= E_LutMode.eAnalogToPhisical;

UW_2_Diameter.stLutDataParam.arrAnalog[0]		:= 0;
UW_2_Diameter.stLutDataParam.arrPhisical[0]		:= 200;	//[mm]
UW_2_Diameter.stLutDataParam.arrAnalog[1]		:= 2600;
UW_2_Diameter.stLutDataParam.arrPhisical[1]		:= 355;	//[mm]	
UW_2_Diameter.stLutDataParam.arrAnalog[2]		:= 7500;
UW_2_Diameter.stLutDataParam.arrPhisical[2]		:= 97;	//[mm]	
UW_2_Diameter.stLutDataParam.arrAnalog[3]		:= 32000;
UW_2_Diameter.stLutDataParam.arrPhisical[3]		:= 0;	

UW_2_Diameter.Diameter_Unfiltred 
			:= LookUP_Table(RawValue:=gMachineCtrl.IO.In.UW_2_Diameter,pDataParam:= ADR(UW_2_Diameter.stLutDataParam));	
			
IF gMachineCtrl.Parameters.UW_2_Param.ForceDiameter THEN
	UW_2_Diameter.Diameter_filtred := gMachineCtrl.Parameters.UW_2_Param.ForcedDiameter;
ELSE
	UW_2_Diameter.DiameterLPF(IN:=UW_2_Diameter.Diameter_Unfiltred,out=> UW_2_Diameter.Diameter_filtred);	
END_IF
END_ACTION

ACTION ACT_GearRatio:


	IF (UW_1_Diameter.Diameter_filtred  > 0) THEN																		
	//	UW_1_Data.CalculatedRotSpeed	:= (gMachineCtrl.Parameters.WebLinarSpeed * 360)/ (UW_1_Diameter.Diameter_filtred * PI);
		IF gMachineCtrl.Cmd.UW_1_Cmd.JogFwd THEN
			UW_1_Data.CalculatedGear	:= (gMachineCtrl.Parameters.WebLinarSpeed )/ (UW_1_Diameter.Diameter_filtred * PI);
		ELSIF gMachineCtrl.Cmd.UW_1_Cmd.JogSFwdSlow THEN
			UW_1_Data.CalculatedGear	:= (gMachineCtrl.Parameters.WebLinarSpeedSlow )/ (UW_1_Diameter.Diameter_filtred * PI);
		ELSIF gMachineCtrl.Cmd.UW_1_Cmd.JogBack THEN
			UW_1_Data.CalculatedGear	:= (-gMachineCtrl.Parameters.WebLinarSpeed )/ (UW_1_Diameter.Diameter_filtred * PI);
		ELSIF gMachineCtrl.Cmd.UW_1_Cmd.JogBackdSlow THEN
			UW_1_Data.CalculatedGear	:= (-gMachineCtrl.Parameters.WebLinarSpeedSlow )/ (UW_1_Diameter.Diameter_filtred * PI);			
		ELSE
			UW_1_Data.CalculatedGear	:= 0;
		END_IF
	END_IF
	
	gWebAxes.UW_1.Crtl.MultiAxis.Input.Parameter.GearInMultiMaster.GearRatio1:=UW_1_Data.CalculatedGear;
	gWebAxes.UW_1.Crtl.MultiAxis.Input.Parameter.GearInMultiMaster.GearRatio2:=UW_1_Data.Tension.TensionGear;
	gWebAxes.UW_1.Crtl.MultiAxis.Input.Parameter.GearInMultiMaster.GearRatio3:=UW_1_Data.Dancer.DancerGear;
	
	
	IF (UW_2_Diameter.Diameter_filtred  > 0) THEN																		
	//	UW_1_Data.CalculatedRotSpeed	:= (gMachineCtrl.Parameters.WebLinarSpeed * 360)/ (UW_1_Diameter.Diameter_filtred * PI);
		IF gMachineCtrl.Cmd.UW_2_Cmd.JogFwd THEN
			UW_2_Data.CalculatedGear	:= (gMachineCtrl.Parameters.WebLinarSpeed )/ (UW_2_Diameter.Diameter_filtred * PI);
		ELSIF gMachineCtrl.Cmd.UW_2_Cmd.JogSFwdSlow THEN
			UW_2_Data.CalculatedGear	:= (gMachineCtrl.Parameters.WebLinarSpeedSlow )/ (UW_2_Diameter.Diameter_filtred * PI);
		ELSIF gMachineCtrl.Cmd.UW_2_Cmd.JogBack THEN
			UW_2_Data.CalculatedGear	:= (-gMachineCtrl.Parameters.WebLinarSpeed )/ (UW_2_Diameter.Diameter_filtred * PI);
		ELSIF gMachineCtrl.Cmd.UW_2_Cmd.JogBackdSlow THEN
			UW_2_Data.CalculatedGear	:= (-gMachineCtrl.Parameters.WebLinarSpeedSlow )/ (UW_2_Diameter.Diameter_filtred * PI);			
		ELSE
			UW_2_Data.CalculatedGear	:= 0;
		END_IF
	END_IF
	
	gWebAxes.UW_2.Crtl.MultiAxis.Input.Parameter.GearInMultiMaster.GearRatio1:=UW_2_Data.CalculatedGear;	
	gWebAxes.UW_2.Crtl.MultiAxis.Input.Parameter.GearInMultiMaster.GearRatio2:=UW_2_Data.Tension.TensionGear;
	gWebAxes.UW_2.Crtl.MultiAxis.Input.Parameter.GearInMultiMaster.GearRatio3:=UW_2_Data.Dancer.DancerGear;
END_ACTION

ACTION ACT_init:
UW_1_Diameter.DiameterLPF.Fc:=1;
UW_2_Diameter.DiameterLPF.Fc:=1;


UW_1_Data.Tension.LoadCellLPF.Fc:=15;
UW_2_Data.Tension.LoadCellLPF.Fc:=15;

UW_1_Data.Dancer.DancerLPF.Fc:=1;
UW_2_Data.Dancer.DancerLPF.Fc:=1;


// UW1 Tension loop
UW_1_Data.Tension.FB_TensionLoop.Kp	:= 0.1;
UW_1_Data.Tension.FB_TensionLoop.Tn	:= T#0MS;
UW_1_Data.Tension.FB_TensionLoop.Td	:= T#0MS;
UW_1_Data.Tension.FB_TensionLoop.PidOutMaxValue	:= 1000;
UW_1_Data.Tension.FB_TensionLoop.PidOutMinValue	:= -1000;
UW_1_Data.Tension.FB_TensionLoop.Hold			:= FALSE;

// UW2 Tension loop
UW_2_Data.Tension.FB_TensionLoop.Kp	:= 0.1;
UW_2_Data.Tension.FB_TensionLoop.Tn	:= T#0MS;
UW_2_Data.Tension.FB_TensionLoop.Td	:= T#0MS;
UW_2_Data.Tension.FB_TensionLoop.PidOutMaxValue	:= 1000;
UW_2_Data.Tension.FB_TensionLoop.PidOutMinValue	:= -1000;
UW_2_Data.Tension.FB_TensionLoop.Hold			:= FALSE;
END_ACTION

ACTION ACT_MotionFBcall:


	UW_1_AxisFB(AxisCtrlPtr:=ADR(gWebAxes.UW_1.Crtl.Basic_axis),AxisRef:= gWebAxes.UW_1.Ref);
	
	UW_1_MultiAxisFB(AxisRef := gWebAxes.UW_1.Ref ,MasterRef := gWebAxes.UwVmaster.Ref,
							MasterRef2 := gWebAxes.UwVmaster.Ref,MasterRef3 := gWebAxes.UwVmaster.Ref, MasterRef4 := gWebAxes.UwVmaster.Ref,
							BasicAxisCtrlPtr := ADR(gWebAxes.UW_1.Crtl.Basic_axis), 
							MultiAxisCtrlPtr := ADR(gWebAxes.UW_1.Crtl.MultiAxis));
	
	UW_2_AxisFB(AxisCtrlPtr:=ADR(gWebAxes.UW_2.Crtl.Basic_axis),AxisRef:= gWebAxes.UW_2.Ref);
	
	UW_2_MultiAxisFB(AxisRef := gWebAxes.UW_2.Ref ,MasterRef := gWebAxes.UwVmaster.Ref,
							MasterRef2 := gWebAxes.UwVmaster.Ref,MasterRef3 := gWebAxes.UwVmaster.Ref, MasterRef4 := gWebAxes.UwVmaster.Ref,
							BasicAxisCtrlPtr := ADR(gWebAxes.UW_2.Crtl.Basic_axis), 
							MultiAxisCtrlPtr := ADR(gWebAxes.UW_2.Crtl.MultiAxis));

							
	Output_AxisFB(AxisCtrlPtr:=ADR(gWebAxes.Output.Crtl.Basic_axis),AxisRef:= gWebAxes.Output.Ref);
	

						
	UwVmaster_AxisFB(AxisCtrlPtr:=ADR(gWebAxes.UwVmaster.Crtl.Basic_axis),AxisRef:= gWebAxes.UwVmaster.Ref);
END_ACTION

ACTION ACT_Tension_1:

////////////UW1
UW_1_Data.Tension.stLutDataParam.eLutMode	:= E_LutMode.eAnalogToPhisical;


UW_1_Data.Tension.stLutDataParam.arrAnalog[0]		:= -3700;//-30000;
UW_1_Data.Tension.stLutDataParam.arrPhisical[0]		:= 0;//11000;	//[Dummy]
UW_1_Data.Tension.stLutDataParam.arrAnalog[1]		:= 12700;//-11500;
UW_1_Data.Tension.stLutDataParam.arrPhisical[1]		:= 300;//10000;	//[gram]	
UW_1_Data.Tension.stLutDataParam.arrAnalog[2]		:= 35500;//-600;
UW_1_Data.Tension.stLutDataParam.arrPhisical[2]		:= 700;//0;	//[gram]	
UW_1_Data.Tension.stLutDataParam.arrAnalog[3]		:= 65535;//20000;
UW_1_Data.Tension.stLutDataParam.arrPhisical[3]		:= 1500;//2000;	//[Dummy]


UW_1_Data.Tension.Tension_Unfiltred
			:= LookUP_Table(RawValue:=gMachineCtrl.IO.In.UW_1_LoacCell,pDataParam:= ADR(UW_1_Data.Tension.stLutDataParam));	

UW_1_Data.Tension.LoadCellLPF(IN:=UW_1_Data.Tension.Tension_Unfiltred,out=> UW_1_Data.Tension.Tension_filtred);	
	
UW_1_Data.Tension.FB_TensionLoop.Kp			:= gMachineCtrl.Parameters.UW_1_Param.kp;
UW_1_Data.Tension.FB_TensionLoop.Tn			:= gMachineCtrl.Parameters.UW_1_Param.TN;
UW_1_Data.Tension.FB_TensionLoop.Enable			:= gMachineCtrl.Parameters.UW_1_Param.EnableTension;  
UW_1_Data.Tension.FB_TensionLoop.SetTension		:= gMachineCtrl.Parameters.UW_1_Param.SetTension;
UW_1_Data.Tension.FB_TensionLoop.ActTension		:= UW_1_Data.Tension.Tension_filtred;
UW_1_Data.Tension.FB_TensionLoop.Invert			:= TRUE;
UW_1_Data.Tension.FB_TensionLoop();

IF (UW_1_Diameter.Diameter_filtred  > 0) THEN
	UW_1_Data.Tension.TensionGear	:= (UW_1_Data.Tension.FB_TensionLoop.CorrectionSpeed )/ (UW_1_Diameter.Diameter_filtred * PI);
ELSE
	UW_1_Data.Tension.TensionGear	:=0;
END_IF
END_ACTION

ACTION ACT_Tension_2:

////////////UW2
UW_2_Data.Tension.stLutDataParam.eLutMode	:= E_LutMode.eAnalogToPhisical;


UW_2_Data.Tension.stLutDataParam.arrAnalog[0]		:= -5000;//-30000;
UW_2_Data.Tension.stLutDataParam.arrPhisical[0]		:= 0;//11000;	//[Dummy]
UW_2_Data.Tension.stLutDataParam.arrAnalog[1]		:= 6000;//-11500;
UW_2_Data.Tension.stLutDataParam.arrPhisical[1]		:= 300;//10000;	//[gram]	
UW_2_Data.Tension.stLutDataParam.arrAnalog[2]		:= 20000;//-600;
UW_2_Data.Tension.stLutDataParam.arrPhisical[2]		:= 700;//0;	//[gram]	
UW_2_Data.Tension.stLutDataParam.arrAnalog[3]		:= 65535;//20000;
UW_2_Data.Tension.stLutDataParam.arrPhisical[3]		:= 1500;//2000;	//[Dummy]


UW_2_Data.Tension.Tension_Unfiltred
			:= LookUP_Table(RawValue:=gMachineCtrl.IO.In.UW_2_LoacCell,pDataParam:= ADR(UW_2_Data.Tension.stLutDataParam));	

UW_2_Data.Tension.LoadCellLPF(IN:=UW_2_Data.Tension.Tension_Unfiltred,out=> UW_2_Data.Tension.Tension_filtred);	
	
UW_2_Data.Tension.FB_TensionLoop.Kp			:= gMachineCtrl.Parameters.UW_2_Param.kp;
UW_2_Data.Tension.FB_TensionLoop.Tn			:= gMachineCtrl.Parameters.UW_2_Param.TN;
UW_2_Data.Tension.FB_TensionLoop.Enable			:= gMachineCtrl.Parameters.UW_2_Param.EnableTension;  
UW_2_Data.Tension.FB_TensionLoop.SetTension		:= gMachineCtrl.Parameters.UW_2_Param.SetTension;
UW_2_Data.Tension.FB_TensionLoop.ActTension		:= UW_2_Data.Tension.Tension_filtred;
UW_2_Data.Tension.FB_TensionLoop.Invert			:= TRUE;
UW_2_Data.Tension.FB_TensionLoop();

IF (UW_2_Diameter.Diameter_filtred  > 0) THEN
	UW_2_Data.Tension.TensionGear	:= (UW_2_Data.Tension.FB_TensionLoop.CorrectionSpeed )/ (UW_2_Diameter.Diameter_filtred * PI);
ELSE
	UW_2_Data.Tension.TensionGear	:= 0;
END_IF
END_ACTION

END_PROGRAM

// ---- POUs/Lib/Signal/LookUP_Table.TcPOU
FUNCTION LookUP_Table : LREAL
VAR_INPUT
	RawValue: 		LREAL;
	pDataParam: 	POINTER TO ST_LookUpTableParam; (*analog value parameter  // arr_X_Param[0] = smallest vaule  arr_X_Param[arr_max] = bigest vaule*)
END_VAR

VAR CONSTANT
	arr_max : INT := 40; (*maximum size of array for look up table*)
END_VAR
VAR
	i : INT;
	Y2 : LREAL;
	Y1 : LREAL;
	X1 : LREAL;
	X2 : LREAL;
	
	j:	INT;
	XY: ARRAY[0..45, 0..1] OF LREAL;
	PointsNum: INT;
	tempLookUP_TableMem:	LREAL;
END_VAR

(*IF pDataParam^.eLutMode = E_LutMode.eDisabled THEN
	LookUP_Table:=	LREAL_TO_LINT(RawValue);
ELSIF pDataParam^.eLutMode = E_LutMode.eAnalogToPhisical THEN  
	FOR i:= 0 TO arr_max - 1 DO
		IF (RawValue >= LINT_TO_LREAL(pDataParam^.arrAnalog[i])) AND RawValue <= (LINT_TO_LREAL(pDataParam^.arrAnalog[i+1])) THEN
			X1 := (LINT_TO_LREAL(pDataParam^.arrAnalog[i])) ;//Analog value
			X2 := (LINT_TO_LREAL(pDataParam^.arrAnalog[i+1])) ;//Analog value
			Y1 := (pDataParam^.arrPhisical[i]) ;//Physics value
			Y2 := (pDataParam^.arrPhisical[i+1]) ;//Physics value			
			LookUP_Table:= LREAL_TO_LINT((Y2 - Y1)/(X2 - X1) * ((RawValue) - X1) + Y1) ;
			EXIT;		 			 	
		END_IF	 	
	END_FOR	
ELSIF pDataParam^.eLutMode = E_LutMode.ePhisicalToAnalog THEN 
	FOR i := 0 TO arr_max - 1 DO
		IF (RawValue >= pDataParam^.arrPhisical[i]) AND RawValue <= (pDataParam^.arrPhisical[i+1]) THEN
			Y1 := (LINT_TO_LREAL(pDataParam^.arrAnalog[i])) ;//Analog value
			Y2 := (LINT_TO_LREAL(pDataParam^.arrAnalog[i+1])) ;//Analog value
			X1 := (pDataParam^.arrPhisical[i]) ;//Physics value
			X2 := (pDataParam^.arrPhisical[i+1]) ;//Physics value			
			LookUP_Table:= LREAL_TO_LINT((Y2 - Y1)/(X2 - X1) * ((RawValue) - X1) + Y1) ;
			EXIT;	
		END_IF
	END_FOR	
END_IF*)
	

//////////////////////////////////////////////////////////////////////
IF pDataParam^.eLutMode = E_LutMode.eAnalogToPhisical THEN  
	FOR i := 0 TO arr_max - 1 DO
		X1 := (LINT_TO_LREAL(pDataParam^.arrAnalog[i])) ;//Analog value
		X2 := (LINT_TO_LREAL(pDataParam^.arrAnalog[i+1])) ;//Analog value
		XY[i,0]:= 	LINT_TO_LREAL(pDataParam^.arrAnalog[i]);
		XY[i,1]:= 	pDataParam^.arrPhisical[i];
		IF (X1 = 0) AND (X2 = 0) THEN 
			PointsNum:=	i;
			EXIT;
		END_IF		
	END_FOR
	
	IF i = arr_max THEN
		PointsNum := arr_max;
	END_IF
	
	IF PointsNum >= 2 THEN				 	
		i := 1;
		WHILE (i < PointsNum) AND (XY[i,0] <= RawValue) DO
			i := i + 1;
		END_WHILE;
		LookUP_Table := ((XY[i,1] - XY[i-1,1]) * RawValue - XY[i,1] * XY[i-1,0] + XY[i-1,1] * XY[i,0]) / (XY[i,0] - XY[i-1,0]);
	ELSE
		LookUP_Table:= RawValue;			
	END_IF
		
ELSIF pDataParam^.eLutMode = E_LutMode.ePhisicalToAnalog THEN 
	FOR i := 0 TO arr_max - 1 DO
		X1 := (pDataParam^.arrPhisical[i]) ;//Physics value
		X2 := (pDataParam^.arrPhisical[i+1]) ;//Physics value
		XY[i,0]:= 	pDataParam^.arrPhisical[i];
		XY[i,1]:= 	LINT_TO_LREAL(pDataParam^.arrAnalog[i]);			
		IF (X1 = 0) AND (X2 = 0) THEN
			PointsNum:=	i;	 
			EXIT;
		END_IF		
	END_FOR	
	
	IF PointsNum >= 2 THEN 				
		i := 1;
		WHILE (i < PointsNum) AND (XY[i,0] <= RawValue) DO
			i := i + 1;
		END_WHILE;
		tempLookUP_TableMem:= ((XY[i,1] - XY[i-1,1]) * RawValue - XY[i,1] * XY[i-1,0] + XY[i-1,1] * XY[i,0]) / (XY[i,0] - XY[i-1,0]);
		LookUP_Table:=	(MIN(XY[(PointsNum-1),1],tempLookUP_TableMem));
	ELSE
		LookUP_Table:=	RawValue;
	END_IF
END_IF

END_FUNCTION

// ---- POUs/App/FB_DancerCtrl.TcPOU
FUNCTION_BLOCK FB_DancerCtrl
VAR_INPUT
	Enable	: BOOL;
	DancerFull:BOOL;
	DancerPosition	:REAL;
	Ctrl_Type	: E_DancerCtrlTyp;
	//Ctrl_ref:				REFERENCE TO Ctrl_Typ;
END_VAR
VAR_OUTPUT
	Jog:BOOL;
	dancerFullStatus:BOOL;
END_VAR
VAR
	FilterOn:TON:=(PT:=T#50MS);
	FilterOff:TON:=(PT:=T#50MS);
	
	PositionMax	: REAL := 200;//mm
	PositionMin	: REAL := 100;//mm
END_VAR


IF Enable THEN
	
	IF Ctrl_Type = E_DancerCtrlTyp.DIGITAL THEN
		ACT_Digital();
	ELSIF Ctrl_Type = E_DancerCtrlTyp.ANALOG	THEN
		ACT_Analog();
	END_IF

ELSE
	Jog := FALSE;
	dancerFullStatus := FALSE;
END_IF

ACTION ACT_Analog:


IF DancerPosition > PositionMax THEN
	Jog := TRUE;
ELSIF
	DancerPosition < PositionMin THEN
	 Jog := FALSE;	
END_IF

 dancerFullStatus := (DancerPosition < PositionMax);
END_ACTION

ACTION ACT_Digital:


	FilterOn(IN:=DancerFull);
	FilterOff(IN:=NOT(DancerFull));

	IF (DancerFull  = TRUE) AND FilterOn.Q  THEN
		Jog:=FALSE;
	ELSIF FilterOff.Q THEN
		Jog:=TRUE;
	END_IF
	
dancerFullStatus := FilterOn.Q;
END_ACTION

END_FUNCTION_BLOCK

// ---- POUs/Lib/FB_TensionLoop.TcPOU
FUNCTION_BLOCK FB_TensionLoop
VAR_INPUT
 Enable:			BOOL;
 SetTension:		REAL;
 ActTension:		REAL;
 Hold:				BOOL;
 Invert:			BOOL;
//	stParams:		ST_CTRL_PID_PARAMS;
 Kp:				LREAL;
 Tn:				TIME;
 Td:				TIME;
 PidOutMaxValue:	LREAL;
 PidOutMinValue:	LREAL;	
	
END_VAR
VAR_OUTPUT
	CorrectionSpeed:	REAL;
END_VAR
VAR
 Error:	REAL;
 PID:				FB_CTRL_PID;
 PidLimiter:		FB_CTRL_LIMITER;
 Pidstparams:		ST_CTRL_PID_PARAMS;
 LimiterstParams:	ST_CTRL_LIMITER_PARAMS;	
	
 fbGetCurTaskIdx: 		GETCURTASKINDEX;
 TaskCycleTimeUDINT: 	UDINT;
 TaskCycleTime: 		TIME;
END_VAR


IF (TaskCycleTimeUDINT = 0) THEN
	fbGetCurTaskIdx();
	TaskCycleTimeUDINT := _TaskInfo[fbGetCurTaskIdx.index].CycleTime;
	TaskCycleTime	:= UDINT_TO_TIME(TaskCycleTimeUDINT/10000); 
END_IF


IF (Enable = FALSE) THEN
	pid.eMode	:= eCTRL_MODE_IDLE;
ELSE
	pid.eMode	:= eCTRL_MODE_ACTIVE;	
END_IF

// Call PID function	

PID.fSetpointValue	:= SetTension; 
PID.fActualValue	:= ActTension; 
PID.bHold			:= Hold;

Pidstparams.fKp	:= Kp; 
Pidstparams.tTn	:= Tn; 
Pidstparams.tTd	:= Td; 
Pidstparams.fOutMaxLimit	:= PidOutMaxValue;
Pidstparams.fOutMinLimit	:= PidOutMinValue;
Pidstparams.tCtrlCycleTime	:= TaskCycleTime; 
Pidstparams.tTaskCycleTime	:= TaskCycleTime;

PID(stParams := Pidstparams);

// Call Limiter function

LimiterstParams.tTaskCycleTime	:= TaskCycleTime;
LimiterstParams.tCtrlCycleTime	:= TaskCycleTime;
LimiterstParams.fMaxOutput		:= Pidstparams.fOutMaxLimit;
LimiterstParams.fMinOutput		:= Pidstparams.fOutMinLimit;

PidLimiter.fIn	:= PID.fOut; 
PidLimiter(stParams := LimiterstParams);

IF (Invert = FALSE) THEN
	CorrectionSpeed	:= LREAL_TO_REAL(PidLimiter.fOut);
ELSE
	CorrectionSpeed	:= LREAL_TO_REAL(- PidLimiter.fOut);	
END_IF

END_FUNCTION_BLOCK

// ---- VISUs/HMI.TcPOU
PROGRAM HMI
VAR
	StartButtonColor:BOOL;
	SwitchOnButtonColor:BOOL;
	StopButtonColor:BOOL;
	LogoRotation:INT;
	ManualLogoRotation:INT;
	EnableManualButton:BOOL;
	
	//Timers color
	TimerColdCutColor:BOOL;
	TimerGripperPostionColor:BOOL;	
	TimerHotWeldColor:BOOL;
	TimerHeaterOnColor:BOOL;	
	StateMotorOnColor:BOOL;		
	TimerGripperopenColor:BOOL;
	TimerGripperRetractColor:BOOL;
	
	//Estop Dialog
	bOpen 						: BOOL;
	fbOpenTrigger 				: R_TRIG;
	bClose 						: BOOL;
	fbCloseTrigger 				: R_TRIG;
	EstopDialogBackgroundColor	: BOOL;
	timerDialogsBackground		:TON;
	
	TC_Restart:TC_Restart;
	
	
	//Scaling 
	onOffScaling : INT := 1000;
	WinderScaling : INT := 1000;
	IOScaling : INT := 1000;
	OutputScaling : INT := 1000;	
	SettingsScaling : INT := 1000;	
	EstopScalling	: INT := 1000;
	
	//INIT
	init:BOOL;
	timerInit:TON;
END_VAR


ACT_init();

IF init THEN
	ACT_Timers();
	IF gMachineCtrl.Simulation = FALSE THEN
		ACT_Dialogs();
	END_IF	
	
	IF gMachineCtrl.Cmd.SwitchOn THEN
		SwitchOnButtonColor := gMachineCtrl.Cmd.SwitchOn ;
	END_IF	
	
	IF gMachineCtrl.Cmd.EmStop THEN
		SwitchOnButtonColor := FALSE ;
	END_IF	
	
	IF FB_Machine_Ctrl.StepNo = 20 THEN
		LogoRotation:= (LogoRotation+5) MOD 360;
	ELSE
		//LogoRotation:=0;
	END_IF
	
	
	IF gMachineCtrl.Cmd.Manual THEN
		ManualLogoRotation:= (ManualLogoRotation+5) MOD 360;
	ELSE
		//LogoRotation:=0;
	END_IF
	
	//EnableManual Button
	IF FB_Machine_Ctrl.StepNo = 10 THEN
		EnableManualButton:=FALSE;
	ELSE
		EnableManualButton:=TRUE;
	END_IF

END_IF

TC_Restart();

ACTION ACT_Dialogs:
bOpen:= (gMachineCtrl.IO.In.E_StopPressed=TRUE);
bClose:= (gMachineCtrl.IO.In.E_StopPressed=FALSE);
//Dialog_1
//Open
fbOpenTrigger(CLK := bOpen);
IF fbOpenTrigger.Q THEN
	OpenDialog('Dialog_Estop',300,200);
END_IF
//Close
fbCloseTrigger(CLK := bClose);
IF fbCloseTrigger.Q THEN
	CloseDialog('Dialog_Estop');
END_IF

timerDialogsBackground(IN:=NOT(timerDialogsBackground.Q),PT:=T#2S);
EstopDialogBackgroundColor:= timerDialogsBackground.ET>T#1S;
END_ACTION

ACTION ACT_init:
timerInit(IN:=TRUE,PT:=T#30S);
init:=timerInit.Q;
END_ACTION

ACTION ACT_Timers:


IF FB_Machine_Run.StepNo = MACHINE_GRIPPER_END_POSITION 
OR FB_Machine_Run.StepNo = MACHINE_GRIPPER_START_POSITION THEN
	TimerGripperPostionColor:=TRUE;
ELSE
	TimerGripperPostionColor:=FALSE;
END_IF


IF FB_Machine_Run.StepNo = MACHINE_COLD_CUT_VALVE_OPEN THEN
	TimerColdCutColor:=TRUE;
ELSE
	TimerColdCutColor:=FALSE;
END_IF

IF FB_Machine_Run.StepNo = MACHINE_WELD_VALVE_OPEN
OR FB_Machine_Run.StepNo = MACHINE_VALVE_CLOSE THEN
	TimerHotWeldColor:=TRUE;
ELSE
	TimerHotWeldColor:=FALSE;
END_IF

IF FB_Machine_Run.FB_HeaterProtection.Busy
OR FB_Machine_Run.StepNo = MACHINE_HEATER_OFF THEN
	TimerHeaterOnColor:=TRUE;
ELSE
	TimerHeaterOnColor:=FALSE;
END_IF

IF FB_Machine_Run.StepNo = MACHINE_GRIPPER_OPEN
OR FB_Machine_Run.StepNo = MACHINE_GRIPPER_CLOSE THEN
	TimerGripperopenColor:=TRUE;
ELSE
	TimerGripperopenColor:=FALSE;
END_IF

IF FB_Machine_Run.StepNo = MACHINE_OUT_GRIPPER_END_POSITION OR FB_Machine_Run.StepNo = MACHINE_OUT_GRIPPER_START_POSITION THEN
	StateMotorOnColor:=TRUE;
ELSE
	StateMotorOnColor:=FALSE;
END_IF

IF FB_Machine_Run.StepNo = MACHINE_GRIPPER_RETRACT
OR FB_Machine_Run.StepNo = MACHINE_GRIPPER_EXCTRACT THEN
	TimerGripperRetractColor:=TRUE;
ELSE
	TimerGripperRetractColor:=FALSE;
END_IF
END_ACTION

END_PROGRAM

// ---- VISUs/infra/OpenDialog.TcPOU
FUNCTION OpenDialog : bool
VAR_INPUT
	sDialogName:STRING;
	iXpos:INT:=0;
	iYpos:INT:=0;
END_VAR
VAR
	stMyRect : VisuElems.VisuStructSimpleRectangle;
	nIteratorSave : INT;
	nCounter : INT;
	pTempClientData : POINTER TO VisuElems.VisuStructClientData;
	pLastClientData : POINTER TO VisuElems.VisuStructClientData;
//general
	iDialogManager : VisuElems.IDialogManager;
	iMessageDialog : VisuElems.IVisualisationDialog;
END_VAR

nIteratorSave := VisuElems.VisuElemBase.Visu_Globals.g_ClientManager.SaveIteration(); 
VisuElems.VisuElemBase.Visu_Globals.g_ClientManager.BeginIteration();

iDialogManager := VisuElems.VisuElemBase.g_VisuManager.GetDialogManager();

// Assign the argument in all currently active clients
pTempClientData := VisuElems.VisuElemBase.Visu_Globals.g_ClientManager.GetNextClient();

WHILE pTempClientData <> 0 DO
	iMessageDialog := iDialogManager.GetDialog(sDialogName); // dialog to be handled is specified
	pLastClientData := pTempClientData;
	pTempClientData := VisuElems.VisuElemBase.g_ClientManager.GetNextClient();
	nCounter := nCounter + 1;
END_WHILE

// Open Dialog on all Clients
iMessageDialog := iDialogManager.GetDialog(sDialogName); // dialog to be handled is specified
IF iMessageDialog <> 0 THEN
	stMyRect.ptTopLeft.iX := iXpos;
	stMyRect.ptTopLeft.iY := iYpos;
	stMyRect.ptBottomRight.iX := 100;
	stMyRect.ptBottomRight.iY := 100;
	iDialogManager.OpenDialog3(iMessageDialog, pLastClientData, TRUE, ADR(stMyRect), 0, VisuElems.Visu_InputFlags.GlobalOpenCloseDialog);
END_IF

VisuElems.VisuElemBase.Visu_Globals.g_ClientManager.RestoreIteration(nIteratorSave);

END_FUNCTION

// ---- VISUs/infra/CloseDialog.TcPOU
FUNCTION CloseDialog : bool
VAR_INPUT
	//pClientData : POINTER TO VisuElems.VisuStructClientData;
	sDialogName:STRING;
END_VAR
VAR
	iDialogManager2 : VisuElems.IDialogManager2 := 0;
	
	pClientData : POINTER TO VisuElems.VisuStructClientData;
	nIteratorSave : INT;
	iDialogManager : VisuElems.IDialogManager;
	iMessageDialog : VisuElems.IVisualisationDialog;
END_VAR


(*dialogMan := VisuElems.g_VisuManager.GetDialogManager();     // the DialogManager is provided via the implicitly available VisuManager

IF dialogMan <> 0 AND pClientData <> 0 THEN
	messageDialog := dialogMan.GetDialog('MessageDialog'); // dialog to be handled is specified
	IF messageDialog <> 0 THEN
		IF (itfDialogManager2 = 0) THEN
			__QUERYINTERFACE(VisuElems.g_VisuManager.GetDialogManager(), itfDialogManager2);
		END_IF
		IF (itfDialogManager2 <> 0) THEN
			itfDialogManager2.CloseDialog2(messageDialog, pClientData, VisuElems.Visu_InputFlags.GlobalOpenCloseDialog);
		ELSE
			dialogMan.CloseDialog(messageDialog, pClientData);	// Closes The Dialog on all "pClientData" 
		END_IF
	END_IF
END_IF*)

nIteratorSave := VisuElems.VisuElemBase.Visu_Globals.g_ClientManager.SaveIteration(); 
VisuElems.VisuElemBase.Visu_Globals.g_ClientManager.BeginIteration();

iDialogManager := VisuElems.VisuElemBase.g_VisuManager.GetDialogManager();

pClientData := VisuElems.VisuElemBase.Visu_Globals.g_ClientManager.GetNextClient();

// Cloase Dialog on all Clients
IF pClientData <> 0 THEN
	iMessageDialog := iDialogManager.GetDialog(sDialogName); // dialog to be handled is specified
	IF iMessageDialog <> 0 THEN
		IF (iDialogManager2 = 0) THEN
			__QUERYINTERFACE(VisuElems.g_VisuManager.GetDialogManager(), iDialogManager2);
		END_IF
		IF (iDialogManager2 <> 0) THEN
			iDialogManager2.CloseDialog2(iMessageDialog, pClientData, VisuElems.Visu_InputFlags.GlobalOpenCloseDialog);
		ELSE
			iDialogManager.CloseDialog(iMessageDialog, pClientData);	// Closes The Dialog on all "pClientData"	
		END_IF
	END_IF
END_IF

VisuElems.VisuElemBase.Visu_Globals.g_ClientManager.RestoreIteration(nIteratorSave);

END_FUNCTION

// ---- POUs/Lib/Inveter_Lib/FB_INV.TcPOU
(*****************************************************************************************
 *  Enverter Oparation FB
 * Author: Dan Naaman
 *****************************************************************************************
 * Implementation of FB
 Actual_Vel_Link- Link to 'vl velocity actual value' From Device IO
 Status_Word_Link- Link to 'Status word' From Device IO
 Set_Vel_Link-Link to 'vl target velocit' From Device IO
 Cntrl_Word_Link-Link to 'Control word' From Device IO
 MasterNetId- Get Value from Ethercat Master In Ethercat Tab
 nSlaveAddr- Get From Actual Drive In Ethercat Tab 'Ethercat Addr' In Device Io
 nIndex,nSubIndex - Get From Actual Drive : In Proccess Data Tab You can Right Click On 'PDO Content'
                    Choose 'Insert' And In dictinarry You can See all Indexes and sub indexes of all
					available Parameters.Once You know The  nIndex,nSubIndex  Click Cancel . 
Env_Status-  shows Current Status Of Inverter .
ResetError- Reset The Error And Set Enable To False :
 *****************************************************************************************)
 
FUNCTION_BLOCK PUBLIC FB_INV
VAR_INPUT
	HWlink:ST_BasicInverter;
	//Set_Vel_Link AT %Q*:INT;
	//INV_Enable:BOOL;
	//ResetError:BOOL;
	ctrl:InverterCtrl_Typ;
	MasterNetId:T_AmsNetID:='15.17.210.19.7.1';
	nSlaveAddr:UINT;
	nSubIndex:BYTE;
	nIndex:WORD;
	
END_VAR
VAR_OUTPUT
	//Actual_Vel_Link AT %I*:INT:=0;
	Error:BOOL;
	ErrorCode:UINT;
	Inv_Status:Enum_INV_Status;
END_VAR
VAR
	//Status_Word_Link AT %I*:UINT;
	//Cntrl_Word_Link AT %Q*:UINT;
	FB_EcCoeSdoRead_DriveError	: FB_EcCoeSdoRead;
	INV_Seq:Enum_INV_Ctrl;
	
	
END_VAR

CASE INV_Seq OF
	Enum_INV_Ctrl.ENV_Disable:
		HWlink.ControlWord:=INT_TO_UINT(Enum_INV_Ctrl.ENV_Disable);
		IF ctrl.Start THEN 
			INV_Seq:=Enum_INV_Ctrl.ENV_GetReady;
		END_IF
	Enum_INV_Ctrl.ENV_GetReady:
		HWlink.ControlWord:=INT_TO_UINT(Enum_INV_Ctrl.ENV_GetReady );
		IF  HWlink.StatusWord =INT_TO_UINT(Enum_INV_Status.ENV_ReadyTo_switchon) THEN 
			INV_Seq:=Enum_INV_Ctrl.ENV_Switch_on;
		END_IF
	Enum_INV_Ctrl.ENV_Switch_on://enable2
		HWlink.ControlWord:=INT_TO_UINT(Enum_INV_Ctrl.ENV_Switch_on);
		IF  HWlink.StatusWord =INT_TO_UINT(Enum_INV_Status.ENV_SwitchedOn) THEN 
			INV_Seq:=Enum_INV_Ctrl.ENV_enable_operation;
		END_IF
	Enum_INV_Ctrl.ENV_enable_operation://enable3
		HWlink.ControlWord:=INT_TO_UINT(Enum_INV_Ctrl.ENV_Enable_operation);  
		IF  HWlink.StatusWord =INT_TO_UINT(Enum_INV_Status.ENV_Operation_Enabled) THEN 
			INV_Seq:=Enum_INV_Ctrl.ENV_Run;
		END_IF
	Enum_INV_Ctrl.ENV_Run:
		IF ctrl.Start =FALSE THEN 
			HWlink.ControlWord:=INT_TO_UINT(Enum_INV_Ctrl.ENV_Disable);
			IF  HWlink.StatusWord =INT_TO_UINT(Enum_INV_Status.ENV_Off) THEN 
				INV_Seq:=Enum_INV_Ctrl.ENV_Disable;
			END_IF
		END_IF
	Enum_INV_Ctrl.ENV_Trip: //error
		IF ctrl.ResetError THEN 
			HWlink.ControlWord:=INT_TO_UINT(Enum_INV_Ctrl.ENV_Reset_Error);
			ctrl.ResetError:=FALSE;
		END_IF
		IF  HWlink.StatusWord =INT_TO_UINT(Enum_INV_Status.ENV_Off) THEN 
			INV_Seq:=0;
			HWlink.ControlWord:=INT_TO_UINT(Enum_INV_Ctrl.ENV_Disable);
			ctrl.Start:=FALSE;
			Error:=FALSE;
			ErrorCode:=0;
		END_IF
		
END_CASE

Error:=HWlink.StatusWord =INT_TO_UINT(Enum_INV_Status.ENV_Trip);
IF Error AND INV_Seq <> Enum_INV_Ctrl.ENV_Trip THEN 
	INV_Seq:=Enum_INV_Ctrl.ENV_Trip;
	FB_EcCoeSdoRead_DriveError.bExecute:=TRUE;
END_IF

Inv_Status:=UINT_TO_INT(HWlink.StatusWord);

FB_EcCoeSdoRead_DriveError(
	sNetId:=MasterNetId , //'169.254.44.60.2.1'
	nSlaveAddr:=1001 , //1001
	nSubIndex:=16#0000 ,//16#0000 
	nIndex:=16#603F , //16#603F
	pDstBuf:=ADR(ErrorCode) , 
	cbBufLen:=SIZEOF(ErrorCode) , 
	bExecute:= , 
	tTimeout:= , 
	bBusy=> , 
	bError=> , 
	nErrId=> );
	
	IF  FB_EcCoeSdoRead_DriveError.bExecute =TRUE AND FB_EcCoeSdoRead_DriveError.bBusy= FALSE THEN 
		 FB_EcCoeSdoRead_DriveError.bExecute:=FALSE;
	END_IF
ctrl.ActualVelocity:=HWlink.ActualSpeed;
HWlink.SetSpeed:=ctrl.SetVelocity;

END_FUNCTION_BLOCK

// ---- POUs/Lib/Motion/SercosAxis/BeckHoff/Beck5xxxAxis_FB.TcPOU
FUNCTION_BLOCK PUBLIC Beck5xxxAxis_FB EXTENDS SercosBasicAxis_FB  
VAR_INPUT		
	io_SafetyState: 		INT;	
END_VAR
VAR_IN_OUT	
END_VAR
VAR_OUTPUT	
END_VAR

VAR
	DebugError					: UINT;
	
END_VAR



SUPER^(AxisRef:=AxisRef);

AxisCtrlPtr^.Output.Status.DriveEnable:=	 NOT (INT_TO_BOOL(io_SafetyState));

METHOD CreateDriveErrMsgDetails : enumMotorEvents
VAR_INPUT
	ErrorId			: UDINT;
END_VAR
CASE ErrorId OF
	 0: 
		CreateDriveErrMsgDetails := enumMotorEvents.NoEvents ;
	16#CD40..16#CD47 :
	
		CreateDriveErrMsgDetails := enumMotorEvents.NoEvents ;
		fnLogMsg(ADR(LogMsg_0),LOG_ERROR,'Beckhoff Drive8 Warning %d',UDINT_TO_DINT(ErrorId),0,0);

 	16#D006: 
		CreateDriveErrMsgDetails := enumMotorEvents.DriveNotReady ;
		fnLogMsg(ADR(LogMsg_0),LOG_ERROR,'ErrorId %d Not Valid',UDINT_TO_DINT(ErrorId),0,0);
	16#D010: 
		CreateDriveErrMsgDetails := enumMotorEvents.DriveNotReady ;
		fnLogMsg(ADR(LogMsg_0),LOG_ERROR,'ErrorId %d Not Ready',UDINT_TO_DINT(ErrorId),0,0);
	16#D011: 
		CreateDriveErrMsgDetails := enumMotorEvents.NoEvents ;
		fnLogMsg(ADR(LogMsg_0),LOG_ERROR,'ErrorId %d Ready',UDINT_TO_DINT(ErrorId),0,0);
	16#D015:
		CreateDriveErrMsgDetails := enumMotorEvents.MotorGeneralError ;
		fnLogMsg(ADR(LogMsg_0),LOG_ERROR,'ErrorId %d Axis error',UDINT_TO_DINT(ErrorId),0,0);
	16#D019:
		CreateDriveErrMsgDetails := enumMotorEvents.MotorGeneralError ;
		fnLogMsg(ADR(LogMsg_0),LOG_ERROR,'ErrorId %d Invalid state',UDINT_TO_DINT(ErrorId),0,0);
	16#D101:
		CreateDriveErrMsgDetails := enumMotorEvents.MotorSupplyError ;	
		fnLogMsg(ADR(LogMsg_0),LOG_ERROR,'ErrorId %d Drive Not Enabled',UDINT_TO_DINT(ErrorId),0,0);
		
	16#D782,16#D783,16#D784:
		CreateDriveErrMsgDetails := enumMotorEvents.MotorFeedBackErr;
		fnLogMsg(ADR(LogMsg_0),LOG_ERROR,'ErrorId %d Endat Encoder Error',UDINT_TO_DINT(ErrorId),0,0);
	16#DCBB:
		CreateDriveErrMsgDetails := enumMotorEvents.DriveComError ;
		fnLogMsg(ADR(LogMsg_0),LOG_ERROR,'ErrorId %d Communication aborted',UDINT_TO_DINT(ErrorId),0,0);

	16#DD42:
		CreateDriveErrMsgDetails := enumMotorEvents.MotorSupplyError;
		fnLogMsg(ADR(LogMsg_0),LOG_ERROR,'ErrorId %d DC link current in limit',UDINT_TO_DINT(ErrorId),0,0);
	16#ED00:
		CreateDriveErrMsgDetails := enumMotorEvents.MotorOverTemp ;
		fnLogMsg(ADR(LogMsg_0),LOG_ERROR,'ErrorId %d Terminal-Overtemperature',UDINT_TO_DINT(ErrorId),0,0);
	
	16#ECD0:
		CreateDriveErrMsgDetails := enumMotorEvents.MotorPositionError ;
		fnLogMsg(ADR(LogMsg_0),LOG_ERROR,'ErrorId %d Positive limit switch warning',UDINT_TO_DINT(ErrorId),0,0);
		
	16#ECD1:
		CreateDriveErrMsgDetails := enumMotorEvents.MotorPositionError ;
		fnLogMsg(ADR(LogMsg_0),LOG_ERROR,'ErrorId %d Neg limit switch warning',UDINT_TO_DINT(ErrorId),0,0);
		
	16#ED01:
		CreateDriveErrMsgDetails := enumMotorEvents.MotorOverCurrent ;
		fnLogMsg(ADR(LogMsg_0),LOG_ERROR,'ErrorId %d Overload - motor',UDINT_TO_DINT(ErrorId),0,0);
	16#ED40:
		CreateDriveErrMsgDetails := enumMotorEvents.MotorOverCurrent ;
		fnLogMsg(ADR(LogMsg_0),LOG_ERROR,'ErrorId %d Internal brake resistor',UDINT_TO_DINT(ErrorId),0,0);
	16#ED41:
		CreateDriveErrMsgDetails := enumMotorEvents.MotorOverCurrent ;
		fnLogMsg(ADR(LogMsg_0),LOG_ERROR,'ErrorId %d External brake resistor',UDINT_TO_DINT(ErrorId),0,0);	
	16#ED42:
		CreateDriveErrMsgDetails := enumMotorEvents.MotorOverCurrent ;
		fnLogMsg(ADR(LogMsg_0),LOG_ERROR,'ErrorId %d Overtemperature - Amplifier',UDINT_TO_DINT(ErrorId),0,0);		
		
	16#ED43:
		CreateDriveErrMsgDetails := enumMotorEvents.MotorSupplyError ;
		fnLogMsg(ADR(LogMsg_0),LOG_ERROR,'ErrorId %d Undervoltage - DC link',UDINT_TO_DINT(ErrorId),0,0);
	16#F2A0:
		CreateDriveErrMsgDetails := enumMotorEvents.DriveComError ;
		fnLogMsg(ADR(LogMsg_0),LOG_ERROR,'ErrorId %d commutation error',UDINT_TO_DINT(ErrorId),0,0);
	16#F2A1,16#F2A3:
		CreateDriveErrMsgDetails := enumMotorEvents.MotorOverCurrent ;
		fnLogMsg(ADR(LogMsg_0),LOG_ERROR,'ErrorId %d Overcurrent error motor',UDINT_TO_DINT(ErrorId),0,0);
		
	16#F2E1:
		CreateDriveErrMsgDetails := enumMotorEvents.MotorSpeedError ;
		fnLogMsg(ADR(LogMsg_0),LOG_ERROR,'ErrorId %d Velocity Control error motor',UDINT_TO_DINT(ErrorId),0,0);
		
	16#F321:
		CreateDriveErrMsgDetails := enumMotorEvents.MotorPositionError  ;
		fnLogMsg(ADR(LogMsg_0),LOG_ERROR,'ErrorId %d  following error Detected',UDINT_TO_DINT(ErrorId),0,0);
 
	16#F324..16#F344:
		CreateDriveErrMsgDetails := enumMotorEvents.MotorPositionError ;
		fnLogMsg(ADR(LogMsg_0),LOG_ERROR,'ErrorId %d Position control - Interpolator error',UDINT_TO_DINT(ErrorId),0,0);
	16#F700..16#FCB4:
		CreateDriveErrMsgDetails := enumMotorEvents.MotorGeneralError ;
		fnLogMsg(ADR(LogMsg_0),LOG_ERROR,'ErrorId %d General Error',UDINT_TO_DINT(ErrorId),0,0);

	16#FCD0,16#FCD1:
		CreateDriveErrMsgDetails := enumMotorEvents.MotorPositionError;
		fnLogMsg(ADR(LogMsg_0),LOG_ERROR,'ErrorId %d limit switch error',UDINT_TO_DINT(ErrorId),0,0);
	16#FCD2,16#FCD3:
		CreateDriveErrMsgDetails := enumMotorEvents.MotorSpeedError;
		fnLogMsg(ADR(LogMsg_0),LOG_ERROR,'ErrorId %d Speed Error',UDINT_TO_DINT(ErrorId),0,0);
	16#FD4B :
		CreateDriveErrMsgDetails := enumMotorEvents.MotorSupplyError;
		fnLogMsg(ADR(LogMsg_0),LOG_ERROR,'ErrorId %d DC link undervoltage',UDINT_TO_DINT(ErrorId),0,0);

	16#FD4C :
		CreateDriveErrMsgDetails := enumMotorEvents.MotorSupplyError;
		fnLogMsg(ADR(LogMsg_0),LOG_ERROR,'ErrorId %d DC link Over voltage',UDINT_TO_DINT(ErrorId),0,0);
		
		
	16#FD51 :
		CreateDriveErrMsgDetails := enumMotorEvents.MotorSupplyError;
		fnLogMsg(ADR(LogMsg_0),LOG_ERROR,'ErrorId %d Power supply phase error',UDINT_TO_DINT(ErrorId),0,0);
		
	16#FDD3 :
		CreateDriveErrMsgDetails := enumMotorEvents.DriveNotEnabled;
		fnLogMsg(ADR(LogMsg_0),LOG_ERROR,'ErrorId %d Safety switch off while the axis was enabled.',UDINT_TO_DINT(ErrorId),0,0);
	ELSE
		fnLogMsg(ADR(LogMsg_0),LOG_ERROR,'unknown ErrorId %d ',UDINT_TO_DINT(ErrorId),0,0);
		CreateDriveErrMsgDetails := enumMotorEvents.MotorGeneralError;
END_CASE
END_METHOD

END_FUNCTION_BLOCK

// ---- POUs/Lib/Motion/SercosAxis/SercosBasicAxis_FB.TcPOU
FUNCTION_BLOCK PUBLIC SercosBasicAxis_FB EXTENDS BasicAxis_FB  
VAR_INPUT
	io_Class1diagnostic: 	INT;		// (C1D) s-0-11 S-0-135
END_VAR
VAR_IN_OUT
	
END_VAR

VAR_OUTPUT
	
END_VAR
VAR
	FB_EcSoeRead_0 		: FB_EcSoeRead ;
	FB_EcSoeWrite_0		: FB_EcSoeWrite ;
	SercosDrive_Ctrl_Adr: SercosDrive_Ctrl_Adr_typ;
	InitIdnsAdr: BOOL := FALSE;
	SercosDriveDeviceError	: BOOL;
	DiagnosticTON  				: TON;
	
END_VAR



AxisCtrlPtr^.Input.Parameter.Drive.eDriveType := enumDriveType.e5xxxBeckhoff;	
AxisCtrlPtr^.Input.Parameter.Drive.VendorNameID := eVendorNameID.Beckhoff;

SercosDriveDeviceError	:= io_Class1diagnostic.13;

IF InitIdnsAdr = FALSE THEN
	GetIdns();
	InitIdnsAdr := TRUE;
END_IF


{warning disable C0371}
 SUPER^(AxisRef:=AxisRef);
{warning restore C0371}

METHOD CreateDriveErrMsgDetails : enumMotorEvents
VAR_INPUT
		ErrorId			: UDINT;		
END_VAR
fnLogMsg(ADR(LogMsg_0),LOG_ERROR,'ErrorId %d ',ErrorId,0,0);
//Etz to do
CreateDriveErrMsgDetails := enumMotorEvents.NoEvents;
END_METHOD

METHOD DriveErrorHandling : BOOL

VAR
	Error : BOOL;
END_VAR

VAR_INST
	ErrHandState	: INT;
	FB_SoEReset_0	: FB_SoEReset;
	FB_EcSoERead_DriveError		: FB_EcSoERead;
	tmpDriveErrorId				: UDINT;

	MC_Reset_0					: MC_Reset;
	
	tmpErrorEntry			: Eh_ErrorEntry_typ;
END_VAR


CASE ErrHandState OF
	0: // logic init

			ErrHandState	 := 100;
			DiagnosticTON.PT := T#2S;
	
	//************************* Sercos Logic **********************************************
	100: // wait errors	
		IF AxisRef.Status.DriveDeviceError OR SercosDriveDeviceError THEN
			FB_SoEReset_0.Execute				:= FALSE;
			FB_EcSoERead_DriveError.bExecute	:= FALSE;
			ErrHandState	:= 110;
		ELSIF AxisRef.NcToPlc.ErrorCode <> 0 
			AND AxisRef.NcToPlc.ErrorCode <> 18000 THEN
			ErrHandState	:= 300;
		ELSIF AxisCtrlPtr^.Output.Error.fbErrorHandler.EntriesCount > 0 THEN
			// do nothing
			DiagnosticTON.IN := TRUE;
		ELSE	
			DiagnosticTON.IN := TRUE;
		END_IF
		
	(*	IF DiagnosticTON.Q THEN
			IF Meth_ReadDiagnostic(TRUE,Error => Error) THEN
				 IF Error THEN
					FB_SoEReset_0.Execute				:= FALSE;
					FB_EcSoERead_DriveError.bExecute	:= FALSE;
					ErrHandState	:= 110;
				 END_IF
				 DiagnosticTON.IN := FALSE;
				 Meth_ReadDiagnostic(FALSE);
			END_IF
		ELSE
			Meth_ReadDiagnostic(FALSE);
		END_IF	*)
		

		IF ErrHandState <> 100 THEN
			DiagnosticTON.IN := FALSE;
		END_IF
		
	110: // read sercos drive error
		FB_EcSoERead_DriveError.sNetId		:= strEcNetId;
		FB_EcSoERead_DriveError.nSlaveAddr	:= AxisCtrlPtr^.Input.Parameter.Drive.EtherCatAddr;
		FB_EcSoERead_DriveError.pDstBuf		:= ADR(tmpDriveErrorId);
		FB_EcSoERead_DriveError.cbBufLen		:= SIZEOF(tmpDriveErrorId);
		FB_EcSoERead_DriveError.nDriveNo		:= 0;
		FB_EcSoERead_DriveError.nElement		:= EC_SOE_ELEMENT_VALUE;		
		FB_EcSoERead_DriveError.nIdn			:= S_0_IDN+SercosDrive_Ctrl_Adr.DriveError;
		FB_EcSoERead_DriveError.bExecute		:= TRUE;
		
		ErrHandState	:= 111;
	111:
		IF NOT FB_EcSoERead_DriveError.bBusy THEN
			FB_EcSoERead_DriveError.bExecute		:= FALSE;
			IF NOT FB_EcSoERead_DriveError.bError THEN
				// Add Drive Error to ErrorHandler
				tmp_ErrorEntry.ErrorId		:= tmpDriveErrorId;
				tmp_ErrorEntry.ErrorText	:= 'Drive ErrorID: ';
				tmp_ErrorEntry.ErrorText	:= CONCAT(tmp_ErrorEntry.ErrorText, UDINT_TO_STRING(tmp_ErrorEntry.ErrorId));
				tmp_ErrorEntry.ErrorText	:= CONCAT(tmp_ErrorEntry.ErrorText, ', Or 0x');
				tmp_ErrorEntry.ErrorText	:= CONCAT(tmp_ErrorEntry.ErrorText, UDINT_TO_HEX_STRING(tmp_ErrorEntry.ErrorId));
				tmp_ErrorEntry.MotorEvents  := CreateDriveErrMsgDetails(tmp_ErrorEntry.ErrorId);
				AxisCtrlPtr^.Output.Error.fbErrorHandler.ErrorPush(tmp_ErrorEntry);
				
				ErrHandState	:= 112;	// sercos reset
		
			ELSE
				fnLogMsg(ADR(LogMsg_0),LOG_ERROR,'EcSoERead Error %d ,nIdn %d ' ,UDINT_TO_DINT(FB_EcSoERead_DriveError.nErrId),FB_EcSoERead_DriveError.nIdn,0);
				ErrHandState	:= 110;	// read one more time
			END_IF
		END_IF
	112: // wait speed decrease
		IF AxisCtrlPtr^.Output.monitor.ActVelocity < 500 THEN
			ErrHandState	:= 120;	// sercos reset
		END_IF
		
	120: // SercosReset
		FB_SoEReset_0.NetId:= AxisCtrlPtr^.Input.Parameter.pcNetId;
		FB_SoEReset_0.Timeout:= T#10S;
		FB_SoEReset_0.Execute:= TRUE;
		
		ErrHandState	:= 121;
		
	121: // wait sercos reset done
		IF AxisRef.Status.DriveDeviceError = FALSE THEN
			FB_SoEReset_0.Execute	:= FALSE;
			
			ErrHandState	:= 300;
			
		END_IF
		

	300: // Run MC_Reset
		MC_Reset_0.Execute	:= TRUE;
		ErrHandState		:= 301;
	301:
		IF MC_Reset_0.Done 
			AND AxisRef.NcToPlc.ErrorCode = 0
			(*AND Axis.Status.DriveDeviceError = FALSE*) THEN
			MC_Reset_0.Execute	:= FALSE;
	
			ErrHandState	:= 0;
		
		ELSIF MC_Reset_0.Error THEN
			MC_Reset_0.Execute	:= FALSE;
			// Add FB Error to ErrorHandler
			tmp_ErrorEntry.ErrorId		:= MC_Reset_0.ErrorID;
			tmp_ErrorEntry.ErrorText	:= 'FB MC_Reset_0 ErrorID: ';
			tmp_ErrorEntry.ErrorText	:= CONCAT(tmp_ErrorEntry.ErrorText, UDINT_TO_STRING(tmp_ErrorEntry.ErrorId));
			AxisCtrlPtr^.Output.Error.fbErrorHandler.ErrorPush(tmp_ErrorEntry);
			
			ErrHandState	:= 0;
		END_IF
		
		IF (AxisCtrlPtr^.Output.Status.CommunicationError = TRUE) THEN
			MC_Reset_0.Execute	:= FALSE;
			ErrHandState		:= 400;	
		END_IF
		
	400:
		IF (AxisCtrlPtr^.Output.Status.CommunicationError = FALSE) THEN
			ErrHandState	:= 300;	
		END_IF
		
END_CASE
DiagnosticTON();

FB_EcSoERead_DriveError();
{warning disable C0371}
FB_SoEReset_0(Axis:= AxisRef);
MC_Reset_0(Axis:= AxisRef);
{warning restore C0371}
END_METHOD

METHOD GetIdns : BOOL
VAR_INPUT
END_VAR


VAR
	
	
END_VAR
SercosDrive_Ctrl_Adr.DriveError := 390;
SercosDrive_Ctrl_Adr.Diagnostic := 13;
END_METHOD

METHOD Meth_ReadDiagnostic : BOOL
VAR_INPUT
	Execute: BOOL;
END_VAR

VAR_INST
	ReadDiagState : INT;
	ReadDiagTrig: Trigger;
	
	Diagnostic  				: UINT;

END_VAR

VAR_OUTPUT
	Error: BOOL;
END_VAR

IF ReadDiagTrig.EDGEPOS(Execute) THEN
	ReadDiagState := 1;
END_IF


IF ReadDiagTrig.EDGENEG(Execute) THEN
	ReadDiagState := 1;
END_IF



CASE ReadDiagState OF
	0:
		FB_EcSoeRead_0.bExecute := FALSE;	
	1:
	
		IF DiagnosticTON.Q THEN
			 FB_EcSoeRead_0.sNetId		:= strEcNetId;
			 FB_EcSoeRead_0.nSlaveAddr	:= AxisCtrlPtr^.Input.Parameter.Drive.EtherCatAddr;
		     FB_EcSoeRead_0.pDstBuf		:= ADR(Diagnostic);
		     FB_EcSoeRead_0.cbBufLen		:= SIZEOF(Diagnostic);
		     FB_EcSoeRead_0.nDriveNo		:= 0;
		     FB_EcSoeRead_0.nElement		:= EC_SOE_ELEMENT_VALUE;		
		     FB_EcSoeRead_0.nIdn			:= S_0_IDN+SercosDrive_Ctrl_Adr.Diagnostic;
		     FB_EcSoeRead_0.bExecute		:= TRUE;
			 ReadDiagState := ReadDiagState +1;
		END_IF
	2:
		IF NOT FB_EcSoeRead_0.bBusy THEN
			FB_EcSoeRead_0.bExecute		:= FALSE;
			IF NOT FB_EcSoeRead_0.bError THEN
				ReadDiagState := ReadDiagState +1;
		
			ELSE
				fnLogMsg(ADR(LogMsg_0),LOG_ERROR,'EcSoERead Error %d ,nIdn %d ' ,UDINT_TO_DINT(FB_EcSoeRead_0.nErrId),FB_EcSoeRead_0.nIdn,0);
				ReadDiagState	:= 0;	// read one more time
			END_IF
		END_IF
	3: // MSG parsing bit 13
		IF Diagnostic.13 = TRUE THEN
			Error	:= TRUE;
		END_IF	
		Meth_ReadDiagnostic := TRUE;

END_CASE
END_METHOD

METHOD PRIVATE ReadActualTorque : LREAL
VAR_INPUT
END_VAR
VAR_INST
	ReadTorqueState	: INT;		
	tmp_ActualTorque			: LREAL;
	p92							: REAL	:= 6.22;
END_VAR
(*

CASE ReadTorqueState OF 
	
	0: 
		
		IF THIS^.TorqueReadEnable THEN
			ReadTorqueState	:= 100;
		END_IF
				
	100: // Sercos Over Ethercat
	
		IF THIS^.AxisRexrothTyp THEN
			ReadTorqueState	:= 150;
		ELSE
			ReadTorqueState	:= 110;
		END_IF
	110:
		ReadTorqueState	:= 150;
	150:
		IF THIS^.AxisRexrothTyp THEN
			tmp_ActualTorque	:= INT_TO_LREAL(io_ActualTorque) / 100.0;
		ELSE
			tmp_ActualTorque	:= p92/1000.0 * INT_TO_LREAL(io_ActualTorque) * TorqueConstant;
		END_IF
END_CASE
*)
ReadActualTorque	:= tmp_ActualTorque;
END_METHOD

METHOD ReadDriveError
VAR_INPUT
END_VAR
VAR_INST 
	ErrIdIndex	: WORD;
END_VAR
DriveError := AxisRef.NcToPlc.StateDWord AND 16#10000000 ;
//AxisRef.Status.DriveDeviceError ; //this flag can be used to monitor an drive error

//=======================================================================================================\\	
	ErrIdIndex	:= 16#603F;

//=======================================================================================================\\		


//=============================================EcSoERead==========================================================\\			

 //works somehow
		
	CASE driveReadErrorState OF 
		0:
			IF AxisRef.Status.DriveDeviceError  AND DriveErrorID = 0 AND NOT (FB_EcSoERead_0.bError = TRUE)
				AND NOT SercosReadDriveErrorIdDone  THEN
					driveReadErrorState := 1 ;
			END_IF

		1:
			FB_EcSoERead_0.sNetId		:= AxisCtrlPtr^.Input.Parameter.ecNetId;
			FB_EcSoERead_0.nSlaveAddr	:= AxisCtrlPtr^.Input.Parameter.Drive.EtherCatAddr;
			FB_EcSoERead_0.pDstBuf		:= ADR(DriveErrorID);
			FB_EcSoERead_0.cbBufLen		:= SIZEOF(DriveErrorID);
			FB_EcSoERead_0.nDriveNo		:= 0;
			FB_EcSoERead_0.nElement		:= EC_SOE_ELEMENT_VALUE;		
			FB_EcSoERead_0.nIdn			:= S_0_IDN+390;
			FB_EcSoERead_0.bExecute		:= TRUE;
			FB_EcSoERead_0();
			
			driveReadErrorState := 2 ;
		2:
			SercosReadDriveErrorIdDone := NOT FB_EcSoERead_0.bBusy ;
			IF SercosReadDriveErrorIdDone THEN
				driveReadErrorState := 0 ;
			END_IF
		
			//AxisState := BASIC_STATE_ERROR;	
			
	END_CASE
	
	IF NOT FB_EcSoERead_0.bBusy THEN
	
		FB_EcSoERead_0.sNetId		:= AxisCtrlPtr^.Input.Parameter.ecNetId;
		FB_EcSoERead_0.nSlaveAddr	:=  AxisCtrlPtr^.Input.Parameter.Drive.EtherCatAddr;
		FB_EcSoERead_0.pDstBuf		:= ADR(DriveErrorID);
		FB_EcSoERead_0.cbBufLen		:= SIZEOF(DriveErrorID);
		FB_EcSoERead_0.nDriveNo		:= 0;
		FB_EcSoERead_0.nElement		:= EC_SOE_ELEMENT_VALUE;		
		FB_EcSoERead_0.nIdn			:= S_0_IDN+390;
		FB_EcSoERead_0.bExecute		:= FALSE;
		FB_EcSoERead_0();
	
		IF FB_EcSoERead_0.bError = TRUE THEN
			FB_EcSoERead_0.sNetId		:= AxisCtrlPtr^.Input.Parameter.ecNetId;
			FB_EcSoERead_0.nSlaveAddr	:=  AxisCtrlPtr^.Input.Parameter.Drive.EtherCatAddr;
			FB_EcSoERead_0.pDstBuf		:= ADR(DriveErrorID);
			FB_EcSoERead_0.cbBufLen		:= SIZEOF(DriveErrorID);
			FB_EcSoERead_0.nDriveNo		:= 0;
			FB_EcSoERead_0.nElement		:= EC_SOE_ELEMENT_VALUE;		
			FB_EcSoERead_0.nIdn			:= S_0_IDN+390;
			FB_EcSoERead_0.bExecute		:= TRUE;
			FB_EcSoERead_0();
		END_IF
	
	END_IF

//=======================================================================================================\\	
FB_EcSoERead_0();
END_METHOD

END_FUNCTION_BLOCK

// ---- POUs/Lib/Motion/BasicAxis_FB.TcPOU
FUNCTION_BLOCK PUBLIC BasicAxis_FB// EXTENDS Tc2_EtherCAT_FB 
VAR_INPUT

	AxisCtrlPtr					: POINTER TO Basic_axis_typ ;
	AxisSercosTyp				: BOOL; 
	
	AxisActive						:BOOL := TRUE;
	
	io_HW_State					: UINT;
	io_EtherCatAddr				: WORD;
	io_ActualTemperature		: REAL;
	io_ActualTorque  			: LREAL;
	io_ActualCurrent 			: LREAL;
	io_TorqueLimitPersent 		: UINT;	//[%]
//	io_ActualTorqueReal AT %I* 	: REAL;
//	TorqueConstant				: LREAL; // [Nm/A] depends on drive, only if needed, 1 = if not needed
	ChangeStateLogEnable		: BOOL;
	
END_VAR
VAR_IN_OUT
	AxisRef			: AXIS_REF;
END_VAR

VAR_OUTPUT
	ErrorID			: UDINT ;
	io_TorqueLimit 	: UINT;
END_VAR
VAR
	LogMsgInit			: BOOL := TRUE;
	LogMsg_0 			: LogMsg ;
	
	fbMcPower 			: MC_Power;			// FB for enable and override
	//fbMC_ReadStatus		: MC_ReadStatus;		// FB for Read Statuses
	fbMC_Home			: MC_Home;
	fbMC_Stop			: MC_Stop;
	fbMC_MoveAbs		: MC_MoveAbsolute;
	fbMC_MoveAdd		: MC_MoveAdditive;
	fbMC_MoveRel		: MC_MoveRelative;
	fbMC_MoveVel		: MC_MoveVelocity;
	fbMC_MoveAbs1		: MC_MoveAbsolute;
	fbMC_MoveAdd1		: MC_MoveAdditive;
	fbMC_MoveRel1		: MC_MoveRelative;
	fbMC_MoveVel1		: MC_MoveVelocity;
	fbMC_Jog			: MC_Jog ;
	fbMC_Halt			: MC_Halt;
	fbMC_SetOverride	: MC_SetOverride;
	fbMC_Reset			: MC_Reset;
	FB_EcCoeSdoRead_0 	: FB_EcCoeSdoRead;
	FB_EcCoeSdoWrite_0 	: FB_EcCoeSdoWrite;
	StateCoeSdoRead		: UINT;
	StateCoeSdoWrite	: UINT;	
	
		
	SDOrw				:Tc2_EtherCAT_typ;
	CoeSdoRW			:EcCoeSdo_Ctrl_typ;
	
	rtReadStatusEnable : R_TRIG ;
	rtReadStatusErr : R_TRIG ;
	
	AxisState			: INT;
	LastAxisStep 		: INT ;
	HomingMode			: INT;
	SS_Init				: INT ;
	rtPowerOn			: R_TRIG;

	ErrorTrig  			: Trigger ;
	AbortTrig  			: Trigger ;
	AxisActiveTrig		: Trigger ;
	fbErrorID 			: UDINT ;
	AxisErrorID 		: UDINT ;
	LastErrorID 		: UDINT ;
		
	HomingActive 		: BOOL ;
	InternalPowerHandle : BOOL;
	
	FB_EcCoeSdoRead_Count	: SINT := 0 ;
	//FB_EcCoeSdoRead_0	: FB_EcCoeSdoRead;
	FB_SoEReadDiagNumber_0	: FB_SoEReadDiagNumber;
	//FB_EcSoERead_0	: FB_EcSoERead;
	FB_SoEReset_0		: FB_SoEReset;
	DriveErrorID 		: UDINT ;//DWORD
	DriveError 			: UDINT ;
	
	TempErrorID			: ARRAY[1..100] OF UDINT;
	TempErrorText		: ARRAY[1..100] OF STRING[2048];
	TempErrorIndex		: USINT := 1 ;
	TempLastErrorID		: UDINT ;
	FirstErrorCollectorTrig : Trigger ;
	
	DriveErrorTrig	:Trigger ;
	MC_Reset_counter	: INT;
	
	ErrorAck_Trigger	: Trigger;
	DriveErrorId_ReadOk_CanResetSercos	: BOOL;
	SercosReadDriveErrorIdDone			: BOOL ;
	CanReadDriveErrorIdDone				: BOOL ;
	driveReadErrorState					: INT ;
		
	tmp_ErrorEntry			: Eh_ErrorEntry_typ;
	strEcNetId				: STRING ; (* EtherCAT NetID - String*)

	// Paremters for homing
	State:INT;	
	HomeState:INT;	
	HomeTrig: Trigger;
	Reset:BOOL;	
	Delay:	TON;
	ScalingNumerator :LREAL;
	HomeRefTrig: Trigger;		
	HomingState : INT;
	
	
	ChangeModeOperTrig  : 	Trigger;

	InValidDataFromDrive: BOOL;
	InValidDataFromDriveTrig :Trigger;
	
	NCError18000 : BOOL;
	NCError18000TON: TON;
	
END_VAR

IF LogMsgInit THEN
	LogMsg_0.ptrGlobalArray		:= 	ADR(LogGlobalArray);
	LogMsg_0.ptrEncoderAngle	:= 	ADR(AxisCtrlPtr^.Input.Parameter.PosForLog);	 
	LogMsgInit	:= FALSE;	
END_IF	
LogMsg_0.Enable				:=  AxisCtrlPtr^.Input.Command.LogEnable;
LogMsg_0.logData.category	:=	AxisCtrlPtr^.Input.Parameter.ThreadName;    

AxisCtrlPtr^.Output.Status.Drive.ActiveHW:=	 UINT_TO_BOOL(io_HW_State);
io_TorqueLimit:=	io_TorqueLimitPersent*10;

AxisCtrlPtr^.Input.Parameter.Drive.EtherCatAddr:= WORD_TO_UINT(io_EtherCatAddr);

AxisCtrlPtr^.Output.monitor.SetVelocity:=  	AxisRef.NcToPlc.SetVelo;	

IF NOT AxisCtrlPtr^.Input.Command.Power
	AND AxisCtrlPtr^.Output.Status.AxisInitDone 
		AND AxisCtrlPtr^.Output.Status.FAULT = FALSE 
			AND InternalPowerHandle = FALSE 
			AND InValidDataFromDrive = FALSE
			AND 
			(AxisState <> BASIC_STATE_HOME OR AxisCtrlPtr^.Input.Parameter.HomeOptions.stBasic.HomingOnDrive =FALSE)
			THEN
	AxisState := BASIC_STATE_WAIT ;
END_IF
//0x100 bit comm error
IF (io_HW_State.9 = TRUE) AND AxisCtrlPtr^.Output.Status.Drive.ActiveHW  AND (AxisCtrlPtr^.Output.Status.CommunicationError = FALSE) THEN
	AxisCtrlPtr^.Output.Status.CommunicationError	:= TRUE;
	AxisState := ENTER_ETHERCAT_FAILURE ;	
ELSIF (io_HW_State.9 = FALSE) THEN
	AxisCtrlPtr^.Output.Status.CommunicationError	:= FALSE;	
END_IF	
	

IF (AxisCtrlPtr^.Input.Command.Stop = TRUE) THEN
		IF ((AxisState <> BASIC_STATE_READY) AND (AxisState <> BASIC_STATE_ERROR) AND (AxisState <> BASIC_STATE_STOP)) THEN
			(* reset all FB execute inputs we use *)

			ResetAll_MC_FB();			
			AxisState := BASIC_STATE_STOP;
		END_IF        
	END_IF  

IF InValidDataFromDriveTrig.EDGEPOS(InValidDataFromDrive) THEN
	AddNCError(18005,'InValidDataFromDrive : '); 
	AxisCtrlPtr^.Output.Status.AxisInitDone:= FALSE ;  
END_IF

IF 	AxisCtrlPtr^.Output.Error.ErrorCount <> 0 THEN	
	//LastAxisStep := AxisState ;s
	IF AxisState <> BASIC_STATE_ERROR THEN 
		fnLogMsg(ADR(LogMsg_0),LOG_ERROR,'Enter Error ',0,0,0);	
		AxisState := BASIC_STATE_ERROR;	
	END_IF


ELSIF AxisCtrlPtr^.Input.Command.AxisInit AND AxisState <> BASIC_STATE_ERROR THEN
	AxisCtrlPtr^.Input.Command.AxisInit := FALSE ;
	AxisCtrlPtr^.Output.Status.AxisInitDone := FALSE ;

	IF AxisCtrlPtr^.Output.Status.Drive.eUpdate_Staus <> enum_DriveUpdateStatus.UpDating THEN
		SS_Init := 0 ;
	END_IF
	
	fnLogMsg(ADR(LogMsg_0),LOG_INFO,'Enter Init State',0,0,0);
	AxisState := BASIC_STATE_INIT ;
END_IF
IF AxisCtrlPtr^.Output.Status.AxisStatus.DriveDeviceError THEN 
	AxisCtrlPtr^.Output.Status.AxisInitDone := FALSE ;
	AxisCtrlPtr^.Output.Status.ReadyForCmd := FALSE ;
END_IF

IF AxisActive = FALSE THEN
	AxisState := BASIC_STATE_NOT_ACTIVE ;
END_IF

IF AxisActiveTrig.EDGENEG(AxisActive) THEN
	ResetAll_MC_FB() ;
	fnLogMsg(ADR(LogMsg_0),LOG_INFO,'Axis Not Active',0,0,0);
END_IF

IF AxisActiveTrig.EDGEPOS(AxisActive) THEN
	AxisState := BASIC_STATE_INIT ;
	fnLogMsg(ADR(LogMsg_0),LOG_INFO,'Axis is Active',0,0,0);
END_IF

CASE AxisState OF
	
	BASIC_STATE_INIT:
	
		IF THIS^.INIT() THEN
			AxisState := BASIC_STATE_WAIT;
		END_IF
		
	BASIC_STATE_WAIT:
		
		THIS^.WAIT();
		
	BASIC_STATE_POWER_ON:  (* STATE: Power on *)   
			//THIS^.Power(PowerOn := TRUE);
			IF (AxisCtrlPtr^.Output.Status.MC_Power.Status = TRUE) THEN
				AxisState := BASIC_STATE_READY;
			END_IF
	(******************** READY **********************)
	BASIC_STATE_READY:  (* STATE: Waiting for commands *)
		AxisCtrlPtr^.Output.Status.ReadyForCmd := TRUE ;
		AxisCtrlPtr^.Input.Command.ClearFault := FALSE ;
		IF AxisCtrlPtr^.Input.Command.Power AND NOT AxisCtrlPtr^.Output.Status.MC_Power.Status THEN
			AxisState := BASIC_STATE_POWER_ON;

		ELSIF (AxisCtrlPtr^.Input.Command.Home = TRUE)THEN
			fnLogMsg(ADR(LogMsg_0),LOG_INFO,'Start Homing mode=%d',AxisCtrlPtr^.Input.Parameter.HomeOptions.stBasic.HomeMode,0,0);
			AxisCtrlPtr^.Input.Command.Home 		:= FALSE ;
			AxisCtrlPtr^.Output.Status.MC_Home.Done := FALSE ;
			THIS^.HomeDirect(FALSE);
			THIS^.HomeAbsSwitch(FALSE);
			HomeLagError(FALSE) ;
			HomeLagErrExternFeedBack(FALSE) ;
			HomeRefPulse(FALSE);
			DriveHomeRefPulse(FALSE);
			HomeAbsoluteEncoder(FALSE);
			HomeAbsEncLagError(FALSE);
			
			AxisState := BASIC_STATE_HOME;

		ELSIF (AxisCtrlPtr^.Input.Command.Stop = TRUE) THEN
			AxisCtrlPtr^.Output.Status.MC_Stop.Done := FALSE ;
			AxisState := BASIC_STATE_STOP;

		ELSIF (AxisCtrlPtr^.Input.Command.MoveJogPos = TRUE) THEN
			AxisState := BASIC_STATE_JOG_POSITIVE;

		ELSIF (AxisCtrlPtr^.Input.Command.MoveJogNeg = TRUE) THEN
			AxisState := BASIC_STATE_JOG_NEGATIVE;

		ELSIF (AxisCtrlPtr^.Input.Command.MoveAbsolute = TRUE) THEN
			AxisCtrlPtr^.Input.Command.MoveAbsolute := FALSE;
			AxisCtrlPtr^.Output.Status.MC_MoveAbsolut.Done := FALSE ;
			AxisState := BASIC_STATE_MOVE_ABSOLUTE;

		ELSIF (AxisCtrlPtr^.Input.Command.MoveAdditive = TRUE) THEN
			AxisCtrlPtr^.Output.Status.MC_MoveAdditive.Done := FALSE ;
			AxisCtrlPtr^.Input.Command.MoveAdditive := FALSE;	
			AxisState := BASIC_STATE_MOVE_ADDITIVE;

		ELSIF (AxisCtrlPtr^.Input.Command.MoveRelative = TRUE) THEN
			AxisCtrlPtr^.Output.Status.MC_MoveRelative.Done := FALSE ;
			AxisCtrlPtr^.Input.Command.MoveRelative := FALSE;	
			AxisState := BASIC_STATE_MOVE_RELATIVE;
			
		ELSIF (AxisCtrlPtr^.Input.Command.MoveVelocity = TRUE) THEN
			AxisCtrlPtr^.Output.Status.MC_MoveVelocity.In_Velocity := FALSE ;
			AxisCtrlPtr^.Input.Command.MoveVelocity := FALSE;
			fbMC_MoveVel.Execute := FALSE;
			AxisState := BASIC_STATE_MOVE_VELOCITY;
  
		ELSIF (AxisCtrlPtr^.Input.Command.Halt = TRUE) THEN
			AxisCtrlPtr^.Input.Command.Halt := FALSE ;
			AxisCtrlPtr^.Output.Status.MC_Halt.Done := FALSE ;
			fbMC_Halt.Execute := FALSE;
			AxisState := BASIC_STATE_HALT; 	

		END_IF

	(******************** HOME **********************)
	BASIC_STATE_HOME:  (* STATE: start homing process *)
	
	//IF AxisCtrlPtr^.Output.Status.Drive.ActiveHW THEN 
			CASE AxisCtrlPtr^.Input.Parameter.HomeOptions.stBasic.HomeMode OF
					
				MC_DefaultHoming,(* default homing as defined in the SystemManager encoder parameters *)	           
 				MC_Direct:(* Static Homing forcing position from user reference *)  
				
					IF THIS^.HomeDirect(TRUE) THEN
						THIS^.HomeDirect(FALSE);
						AxisState := BASIC_STATE_READY;
					END_IF
					
    			MC_AbsSwitch:        (* Made in hp - Absolute Switch homing plus Limit switches *)
					 IF AxisCtrlPtr^.Output.Status.Drive.ActiveHW THEN(*Not simulator *)
						IF AxisCtrlPtr^.Input.Parameter.HomeOptions.stBasic.HomingOnDrive THEN
							IF DriveHomeAbsSwitch(TRUE) THEN
								AxisCtrlPtr^.Output.Status.MC_Home.Done := TRUE;
								DriveHomeAbsSwitch(FALSE);
								AxisState := BASIC_STATE_READY;
							ELSE
								AxisCtrlPtr^.Output.Status.MC_Home.Done := FALSE;	
							END_IF
	
						ELSE
							IF HomeAbsSwitch(TRUE) THEN // Good for abs Encoder
								AxisCtrlPtr^.Output.Status.MC_Home.Done := TRUE;
								HomeAbsSwitch(FALSE);
								AxisState := BASIC_STATE_READY;
							ELSE
								AxisCtrlPtr^.Output.Status.MC_Home.Done := FALSE;	
							END_IF
						END_IF
					ELSE
						IF THIS^.HomeDirect(TRUE) THEN
							fnLogMsg(ADR(LogMsg_0),LOG_WARNING ,'There is no link simulate homing',0,0,0);
							THIS^.HomeDirect(FALSE);
							AxisState := BASIC_STATE_READY;
						END_IF
					END_IF	
	
					
    			MC_LimitSwitch:     (* Made in hp - Homing against Limit switches *)
				
   				MC_RefPulse:        (* Made in hp - Homing using encoder Reference Pulse "Zero Mark" *)
					IF AxisCtrlPtr^.Input.Parameter.HomeOptions.stBasic.HomingOnDrive AND AxisCtrlPtr^.Output.Status.Drive.ActiveHW THEN
						IF DriveHomeRefPulse(TRUE) THEN
							AxisCtrlPtr^.Input.Command.Home 		:= FALSE;
							AxisCtrlPtr^.Output.Status.MC_Home.Done := TRUE;
							
							DriveHomeRefPulse(FALSE);
							AxisState := BASIC_STATE_READY;
						ELSE
							AxisCtrlPtr^.Output.Status.MC_Home.Done := FALSE;
						END_IF

					ELSE
						IF HomeRefPulse(TRUE) THEN


							HomeRefPulse(FALSE);
							AxisState := BASIC_STATE_READY;
						END_IF
					END_IF	
					
    			MC_Absolute:         (*   Static Homing forcing position from absolute encoder *)
				
						IF HomeAbsoluteEncoder(TRUE) THEN
							AxisCtrlPtr^.Output.Status.MC_Home.Done := TRUE;
							HomeAbsoluteEncoder(FALSE);
							AxisState := BASIC_STATE_READY;
						END_IF
						
				
   				MC_Block:            (* not implemented - Homing against hardware parts blocking movement *)
						IF AxisCtrlPtr^.Output.Status.Drive.ActiveHW THEN
							IF AxisCtrlPtr^.Input.Parameter.HomeOptions.stBasic.HomingOnDrive THEN
								
								IF DriveHomeLagError(TRUE) THEN
									AxisState := BASIC_STATE_READY;
									DriveHomeLagError(FALSE);
								END_IF 
							ELSE
								IF AxisCtrlPtr^.Input.Parameter.HomeOptions.stBasic.eEncoderType = E_EncoderType.Absolute THEN
									 IF HomeAbsEncLagError(TRUE) THEN		
										HomeAbsEncLagError(FALSE);					
										AxisState := BASIC_STATE_READY;
									END_IF
								ELSE	
									IF HomeLagError(TRUE) THEN		
										HomeLagError(FALSE);					
										AxisState := BASIC_STATE_READY;
									END_IF
								END_IF	
							END_IF							
						ELSE
							IF THIS^.HomeDirect(TRUE) THEN
								fnLogMsg(ADR(LogMsg_0),LOG_WARNING ,'There is no link simulate homing',0,0,0);
								THIS^.HomeDirect(FALSE);
								AxisState := BASIC_STATE_READY;
							END_IF
					END_IF		
						
   				MC_ForceCalibration: (* set the calibration flag without perfomring any motion or changing the position *)
    			MC_ResetCalibration : (* resets the calibration flag without perfomring any motion or changing the position *)
			
			END_CASE	
		

			
	(*	ELSE
			IF THIS^.HomeDirect(TRUE) THEN
				fnLogMsg(ADR(LogMsg_0),LOG_WARNING ,'There is no link simulate homing',0,0,0);
				THIS^.HomeDirect(FALSE);
				AxisState := BASIC_STATE_READY;
			END_IF
		END_IF*)
		IF AxisState = BASIC_STATE_READY AND BASIC_STATE_ERROR <>  AxisState THEN
			AxisCtrlPtr^.Input.Command.Home 		:= FALSE;
			AxisCtrlPtr^.Output.Status.MC_Home.Done := TRUE;
			HomingActive := FALSE;
			fnLogMsg(ADR(LogMsg_0),LOG_INFO,'Home finished Type=%d',AxisCtrlPtr^.Input.Parameter.HomeOptions.stBasic.HomeMode,0,0);
		END_IF
	
	BASIC_STATE_STOP:
	
		IF THIS^.Stop() THEN
			AxisState := BASIC_STATE_READY;
		END_IF
		
	BASIC_STATE_HALT:
	
		fbMC_Halt.Execute := TRUE;
		
		AxisState := BASIC_STATE_READY;
		
	BASIC_STATE_MOVE_ABSOLUTE:
	
		IF NOT fbMC_MoveAbs.Active THEN
			fbMC_MoveAbs.Execute := TRUE;
		ELSE
			fbMC_MoveAbs1.Execute := TRUE;
		END_IF
		
		AxisState := BASIC_STATE_READY;
		
	BASIC_STATE_MOVE_ADDITIVE:
	
		IF NOT fbMC_MoveAdd.Active THEN
			fbMC_MoveAdd.Execute := TRUE;
		ELSE
			fbMC_MoveAdd1.Execute := TRUE;
		END_IF
		
		AxisState := BASIC_STATE_READY;
		
	BASIC_STATE_MOVE_RELATIVE:
	
		IF NOT fbMC_MoveRel.Active THEN
			fbMC_MoveRel.Execute := TRUE;
		ELSE(*IF NOT fbMC_MoveRel1.Active THEN*)
			fbMC_MoveRel1.Execute := TRUE;
		END_IF
		
		AxisState := BASIC_STATE_READY;
	
	BASIC_STATE_MOVE_VELOCITY:
		fbMC_MoveVel.Execute := TRUE;
		AxisState := BASIC_STATE_READY;
		
	BASIC_STATE_JOG_POSITIVE:
	
		IF THIS^.Jog() THEN
			AxisState := BASIC_STATE_READY;
		END_IF
		
	BASIC_STATE_JOG_NEGATIVE:
		IF THIS^.Jog() THEN
			AxisState := BASIC_STATE_READY;
		END_IF		
		
	BASIC_STATE_ERROR:
		AxisCtrlPtr^.Input.Command.Power := FALSE ;
		AxisCtrlPtr^.Output.Status.FAULT := TRUE ;	
		AxisCtrlPtr^.Output.Status.ReadyForCmd := FALSE ;
		IF AxisCtrlPtr^.Input.Command.ErrorAcknowledge  THEN
			AxisCtrlPtr^.Input.Command.ErrorAcknowledge	:= FALSE;
			AxisCtrlPtr^.Output.Error.fbErrorHandler.ErrorPop();
			fnLogMsg(ADR(LogMsg_0),LOG_INFO,'Error pop',0,0,0);
		END_IF	
		
		IF AxisCtrlPtr^.Input.Command.ClearFault = TRUE THEN
			fnLogMsg(ADR(LogMsg_0),LOG_INFO,'sClear fault',0,0,0);
			AxisCtrlPtr^.Input.Command.ClearFault := FALSE ;
			AxisCtrlPtr^.Output.Status.FAULT := FALSE ;
		END_IF
		
		IF AxisCtrlPtr^.Output.Error.ErrorCount = 0 AND AxisCtrlPtr^.Output.Status.FAULT = FALSE AND 
			((io_HW_State = 8) OR (AxisCtrlPtr^.Output.Status.Drive.ActiveHW = FALSE))   THEN
			fnLogMsg(ADR(LogMsg_0),LOG_INFO,'Exit Error State',0,0,0);
			AxisState := BASIC_STATE_WAIT;
		END_IF
		
		(* reset all FB execute inputs we use *)
		THIS^.ResetAll_MC_FB();
		
		
	ENTER_ETHERCAT_FAILURE:
	
		AxisCtrlPtr^.Input.Command.Power := FALSE ;
		AxisCtrlPtr^.Output.Status.FAULT := TRUE ;	
		AxisCtrlPtr^.Output.Status.ReadyForCmd := FALSE ;
		
		tmp_ErrorEntry.ErrorId		:= ErrorId;
	    
		tmp_ErrorEntry.ErrorText	:= 'Ether Cat error';
		
		tmp_ErrorEntry.ErrorText	:= CONCAT(tmp_ErrorEntry.ErrorText, UDINT_TO_STRING(tmp_ErrorEntry.ErrorId));
		tmp_ErrorEntry.ErrorText	:= CONCAT(tmp_ErrorEntry.ErrorText, ' Task: ');
		tmp_ErrorEntry.ErrorText	:= CONCAT(tmp_ErrorEntry.ErrorText, AxisCtrlPtr^.Input.Parameter.ThreadName);	
		tmp_ErrorEntry.ErrorText	:= CONCAT(tmp_ErrorEntry.ErrorText, FC_NcErrorMsg(tmp_ErrorEntry.ErrorId));
	
		IF ErrorId <> 18000 THEN	
			fnLogMsg(ADR(LogMsg_0),LOG_ERROR,tmp_ErrorEntry.ErrorText,0,0,0);	
			
			tmp_ErrorEntry.MotorEvents := CreateNCErrMsgDetails(tmp_ErrorEntry.ErrorId);
			
			AxisCtrlPtr^.Output.Error.fbErrorHandler.ErrorPush(tmp_ErrorEntry);
		ELSE
			NCError18000 := TRUE;
		END_IF
		
		(* reset all FB execute inputs we use *)
		THIS^.ResetAll_MC_FB();
		AxisState := BASIC_STATE_ERROR ;
		
END_CASE

IF (LastAxisStep <> AxisState) AND ChangeStateLogEnable THEN
	fnLogMsg(ADR(LogMsg_0),LOG_INFO,'Cng State CurSt=%d LstSt=%d',AxisState,LastAxisStep,0);
	LastAxisStep := AxisState ;
END_IF	


THIS^.Power(PowerOn := AxisCtrlPtr^.Input.Command.Power OR AxisCtrlPtr^.Output.Status.AxisStatus.ErrorPropagationDelayed);
fbMC_Stop(Axis := AxisRef) ;
fbMC_Halt(Axis := AxisRef) ;


THIS^.ReadStatus(FALSE);

IF NOT HomingActive THEN
	MoveAbs();
	MoveAdd();
	MoveRelative();
	MoveVelo();
END_IF
Halt();

SetOverride();
DriveErrorHandling();	

AxisCtrlPtr^.Output.Error.ErrorCount := UDINT_TO_UINT(AxisCtrlPtr^.Output.Error.fbErrorHandler.EntriesCount);
AxisCtrlPtr^.Output.Error.ErrorEntry := AxisCtrlPtr^.Output.Error.fbErrorHandler.ErrorRead();

//AxisCtrlPtr^.Output.Error.ErrorID	 := tmp_ErrorEntry.ErrorId;
//AxisCtrlPtr^.Output.Error.ErrorText	 := tmp_ErrorEntry.ErrorText;
		
StatusUpdate();
MonitorUpdate();



//fnLogTransfer FUNCTION call
fnLogTransfer(ADR(LogMsg_0));

//InValidDataFromDrive:= AxisRef.NcToPlc.StateDWord.30;

METHOD AddNCError : BOOL
VAR_INPUT
	ErrorId			: UDINT;
	ErrorPrefix     : STRING[100];
END_VAR
IF io_HW_State=8 THEN
	
	tmp_ErrorEntry.ErrorId		:= ErrorId;
	
	tmp_ErrorEntry.ErrorText	:= ErrorPrefix;
	
	tmp_ErrorEntry.ErrorText	:= CONCAT(tmp_ErrorEntry.ErrorText, UDINT_TO_STRING(tmp_ErrorEntry.ErrorId));
	tmp_ErrorEntry.ErrorText	:= CONCAT(tmp_ErrorEntry.ErrorText, ' Task: ');
	tmp_ErrorEntry.ErrorText	:= CONCAT(tmp_ErrorEntry.ErrorText, AxisCtrlPtr^.Input.Parameter.ThreadName);	
	tmp_ErrorEntry.ErrorText	:= CONCAT(tmp_ErrorEntry.ErrorText, FC_NcErrorMsg(tmp_ErrorEntry.ErrorId));
	
	IF ErrorId <> 18000 THEN	
		fnLogMsg(ADR(LogMsg_0),LOG_ERROR,tmp_ErrorEntry.ErrorText,0,0,0);	
		
		tmp_ErrorEntry.MotorEvents := CreateNCErrMsgDetails(tmp_ErrorEntry.ErrorId);
		
		AxisCtrlPtr^.Output.Error.fbErrorHandler.ErrorPush(tmp_ErrorEntry);
	ELSE
		NCError18000 := TRUE;
	END_IF
END_IF
END_METHOD

METHOD DriveErrorHandling : BOOL
 
VAR_INST

END_VAR
END_METHOD

METHOD PROTECTED DriveHomeAbsSwitch : BOOL
VAR_INPUT
	Execute: BOOL;
END_VAR

VAR_INST
	State:INT;	
	HomeTrig: Trigger;
	Reset:BOOL;	
	sensorOn : BOOL ;//satatus of the sensor of the begining of the homing
	sensorOff : BOOL ;//satatus of the sensor of the begining of the homing
END_VAR
VAR
	
END_VAR
END_METHOD

METHOD DriveHomeLagError : BOOL
VAR_INPUT
	Execute: BOOL;
END_VAR

VAR_INST
//	State:INT;	
//	HomeTrig: Trigger;
//	Reset:BOOL;	
//	Delay:	TON;		
END_VAR
VAR
	
END_VAR
END_METHOD

METHOD PROTECTED DriveHomeRefPulse : BOOL
VAR_INPUT
	Execute: BOOL;
END_VAR

VAR_INST

END_VAR
VAR
	
END_VAR
END_METHOD

METHOD DriveUnitsTorqueToRealValue : LREAL
VAR_INPUT
	
	Torque: LREAL;	

END_VAR
DriveUnitsTorqueToRealValue := Torque;
END_METHOD

METHOD PRIVATE Halt : BOOL
VAR_INPUT
	
END_VAR
VAR_INST
	errorTrig : Trigger ;	
END_VAR
	Halt :=  FALSE ;
	fbMC_Halt.Deceleration 	:= AxisCtrlPtr^.Input.Parameter.Deceleration;
	fbMC_Halt.Jerk 			:= AxisCtrlPtr^.Input.Parameter.Jerk;
	fbMC_Halt.Options 		:= AxisCtrlPtr^.Input.Parameter.Options;

	
	//fbMC_Halt.Execute := TRUE;
	//AxisCtrlPtr^.Output.Status.MC_Halt.Done := FALSE ;
	(* if axis is stopped go to ready state *)
	IF (fbMC_Halt.Done = TRUE) THEN
		Halt :=  TRUE ;
		AxisCtrlPtr^.Input.Command.Halt := FALSE;
		AxisCtrlPtr^.Output.Status.MC_Halt.Done := TRUE ;
		fbMC_Halt.Execute := FALSE;
	END_IF
	(* check if error occured *)
	IF errorTrig.EDGEPOS(fbMC_Halt.Error) THEN
		
		// Add FB Error to ErrorHandler
		AddNCError(fbMC_Halt.ErrorID , 'NC Error fbMC_Halt ErrorID: ');	
		
		Halt :=  FALSE ;
		AxisCtrlPtr^.Input.Command.Halt := FALSE;
		fbMC_Halt.Execute := FALSE;
		//AxisState := BASIC_STATE_ERROR;
	END_IF
	
	{warning disable C0371}
	//Warning: Access to VAR_IN_OUT <Var> declared in <POU> from external context <Method/Transition/Property>
	fbMC_Halt(Axis := AxisRef) ;
	{warning restore C0371}
	
	IF fbMC_Halt.CommandAborted THEN
		AxisCtrlPtr^.Input.Command.Halt := FALSE;
		AxisCtrlPtr^.Output.Status.MC_Halt.Done := TRUE ;
		fbMC_Halt.Execute := FALSE;
	END_IF
	
	AxisCtrlPtr^.Output.Status.MC_Halt.Busy 			:= fbMC_Halt.Busy ;
	AxisCtrlPtr^.Output.Status.MC_Halt.CommandAborted 	:= fbMC_Halt.CommandAborted ;
	AxisCtrlPtr^.Output.Status.MC_Halt.Active 			:= fbMC_Halt.Active ;
END_METHOD

METHOD HomeAbsEncLagError : BOOL
VAR_INPUT
	Execute: BOOL;
END_VAR

VAR_INST
	LagErrorState : INT;
	HomingLagErrorTrig: 		Trigger;
	io_TorqueLimitPersent_Mem:	UINT;
	PositionBias:				LREAL;	
END_VAR
Reset:= Execute;
IF HomeTrig.EDGEPOS(Reset) THEN
	Reset:=	FALSE;
	LagErrorState:=1;
	HomingActive:= 	TRUE ;
	AxisCtrlPtr^.Output.Status.MC_Home.Done:= FALSE ;
	fbMC_MoveVel.Execute:= FALSE ;
	fbMC_MoveRel.Execute:= FALSE ;
END_IF

IF Execute THEN
	CASE LagErrorState OF
		
		1:		
						 		
	
			IF WriteNC_AxisBoolParam(MC_AxisParameter:=MC_AxisParameter.EnablePosLagMonitoring,ParamValue:=FALSE) THEN
				LagErrorState:= LagErrorState +1;	
			END_IF
																
		2: 										
			IF AxisCtrlPtr^.Input.Parameter.HomeOptions.stBasic.StartDirection = eHomeModeOption.eNEGATIVE THEN								
				fbMC_MoveVel.Direction:= 	MC_Negative_Direction;  					
			ELSIF AxisCtrlPtr^.Input.Parameter.HomeOptions.stBasic.StartDirection = eHomeModeOption.ePOSITIVE THEN								
				fbMC_MoveVel.Direction:= 	MC_Positive_Direction;										
			END_IF
			
			fbMC_MoveVel.Velocity:= AxisCtrlPtr^.Input.Parameter.HomeOptions.stBasic.SwitchVelo;
	
			fbMC_MoveVel.Execute:= 	TRUE ;
			
			LagErrorState:= LagErrorState + 1;
			
		3: 	
			IF (ABS(AxisCtrlPtr^.Output.monitor.ActLagError) > AxisCtrlPtr^.Input.Parameter.HomeOptions.stLagErr.LagErr) THEN
				LagErrorState:= LagErrorState + 1;	
			END_IF
		
		4:	
			IF Stop() THEN
				LagErrorState:= LagErrorState + 1;
				Delay(IN:=	FALSE);					
			END_IF
					
		5:	
			Delay(IN:=	TRUE,PT:=T#1S);		
			IF Delay.Q THEN
				Delay(IN:=FALSE);	
				LagErrorState:= LagErrorState +1;
			END_IF
				
		6: 
			IF AxisCtrlPtr^.Input.Parameter.HomeOptions.stBasic.StartDirection = eHomeModeOption.eNEGATIVE THEN													
				fbMC_MoveRel.Distance:=		AxisCtrlPtr^.Input.Parameter.HomeOptions.stLagErr.TriggerOffsetPos ;					
			ELSIF AxisCtrlPtr^.Input.Parameter.HomeOptions.stBasic.StartDirection = eHomeModeOption.ePOSITIVE THEN								
				fbMC_MoveRel.Distance:=		AxisCtrlPtr^.Input.Parameter.HomeOptions.stLagErr.TriggerOffsetPos*(-1) ;											
			END_IF
			fbMC_MoveRel.Velocity:= AxisCtrlPtr^.Input.Parameter.HomeOptions.stBasic.TriggerVelo;
			
			fbMC_MoveRel.Execute:= 	TRUE ;
			LagErrorState:= LagErrorState + 1;
	 		
					
		7:	
			IF fbMC_MoveRel.Done THEN
				AxisCtrlPtr^.Output.monitor.stAbsEncoder.BlockOffsetPosition := AxisCtrlPtr^.Output.monitor.ActPosition ;
 
				LagErrorState:= 100;
			END_IF
			
 
																				
		100:			
			AxisCtrlPtr^.Input.Command.Home:= FALSE ;
			HomingActive:= 				FALSE;
			fbMC_Home.Execute:= 		FALSE;
			AxisCtrlPtr^.Output.Status.MC_Home.Done:= TRUE ;
			HomeAbsEncLagError:=	TRUE;
			LagErrorState:= 0;		
	END_CASE

END_IF
 
			
fbMC_MoveVel.Acceleration  	:= AxisCtrlPtr^.Input.Parameter.HomeOptions.stBasic.Acc;  
fbMC_MoveVel.Deceleration  	:= AxisCtrlPtr^.Input.Parameter.HomeOptions.stBasic.Dcc;  
fbMC_MoveVel.Jerk			:= AxisCtrlPtr^.Input.Parameter.HomeOptions.stBasic.Jerk;
fbMC_MoveVel.Options		:= AxisCtrlPtr^.Input.Parameter.Options;
fbMC_MoveVel.BufferMode		:= AxisCtrlPtr^.Input.Parameter.BufferMode;

fbMC_MoveRel.Acceleration  	:= AxisCtrlPtr^.Input.Parameter.HomeOptions.stBasic.Acc; 
fbMC_MoveRel.Deceleration  	:= AxisCtrlPtr^.Input.Parameter.HomeOptions.stBasic.Dcc;
fbMC_MoveRel.Jerk			:= AxisCtrlPtr^.Input.Parameter.HomeOptions.stBasic.Jerk;
fbMC_MoveRel.Options		:= AxisCtrlPtr^.Input.Parameter.Options;
fbMC_MoveRel.BufferMode		:= AxisCtrlPtr^.Input.Parameter.BufferMode;

{warning disable C0371}
//Warning: Access to VAR_IN_OUT <Var> declared in <POU> from external context <Method/Transition/Property>

fbMC_Home(Axis:= AxisRef);	
fbMC_MoveVel(Axis:= AxisRef);
fbMC_MoveRel(Axis:= AxisRef);

fbMC_Stop.Deceleration:= 	AxisCtrlPtr^.Input.Parameter.Deceleration;
fbMC_Stop.Jerk:=			AxisCtrlPtr^.Input.Parameter.Jerk;
fbMC_Stop.Options:= 		AxisCtrlPtr^.Input.Parameter.Options;
fbMC_Stop(Axis := AxisRef) ;
{warning restore C0371}

THIS^.HomingGlobalHandle();
END_METHOD

METHOD HomeAbsoluteEncoder : BOOL
VAR_INPUT
	Execute: BOOL;
END_VAR
VAR_INST
	adsReadFB : ADSRead;
	HomeAbsoluteEncState : INT;	
	PrevHomeAbsoluteEncState : INT;	
	fbReadParam_ScalingFactor:	MC_ReadParameter;
	OffsetPos :LREAL;
END_VAR
IF HomeTrig.EDGEPOS(Execute) THEN
	HomeAbsoluteEncState := 1;
	HomingActive:= 		TRUE ;
	HomeAbsoluteEncoder := FALSE;

END_IF	
	
//
	CASE HomeAbsoluteEncState OF
		1:
			fbMC_Home.Execute:= FALSE;
			HomeAbsoluteEncState := HomeAbsoluteEncState+1;	
		2:
			
